// I/O Inputs              
	IN_MesAlarmPwr_IO		   : BOOL ;	              // (NA)[P,H,B] Remote control Power supply Error IO  	
	MesDataExd					: CB_Switch ; 		
END_VAR

VAR_OUTPUT
	
	//Child objects
	OUT_CmdOpen_IO	           : BOOL ; 	          // (NA) Physical I/O Open Command IO
	OUT_CmdClose_IO			   : BOOL ; 	          // (NA) Physical I/O Close Command IO
	
END_VAR


VAR
	
	//M_OPENCLOSE VARIABLES//

	//M_OPENCLOSE VARIABLES//	
	ParamTP_Open	 			: TP ;				(* (NA) Temporisation for Open pulse Command*)
	ParamTP_Close 				: TP ;				(* (NA) Temporisation for Close pulse Command	*)
		
END_VAR

METHOD M_AlarmManagement
//////////////////
// Manages Contactor alarms and warnings
/////////////////

VAR 
	// Method local variables (reinitialized at each cycle) 
	FB_AlarmCodeManager			: FB_AlarmCodeManager ; 

END_VAR
VAR_INPUT
	
END_VAR
// Check if command and measures are matching after tempo
FB_CheckCommand	(T:= ParamTimeOut_Close, bCmd:=OUT_CmdClose_IO , bMes := MesDataExd.MesData.MesClosed , bImpulsion := FALSE , bReset := CmdClearFault_G OR OUT_CmdClose_IO) ; 
FB_CheckCommand2(T:= ParamTimeOut_Open , bCmd:= OUT_CmdOpen_IO , bMes :=NOT MesDataExd.MesData.MesClosed , bImpulsion := FALSE , bReset := CmdClearFault_G OR OUT_CmdOpen_IO) ; 

TON_NotClosedAndNotOpened(IN:=  NOT MesClosed AND NOT MesOpened , PT := ParamTimeOut_Alarm) ; 
TON_ClosedAndOpened(IN:=MesClosed AND MesOpened, PT := ParamTimeOut_Alarm) ; 

// ALARM CODE //

	FB_AlarmCodeManager(
		bAlarm1			:= FALSE 	, 								// 
		bAlarm2			:= TON_NotClosedAndNotOpened.Q,					// Incoherent State measure (Not Opened and not Closed)
		bAlarm3 		:= TON_ClosedAndOpened.Q   , 					// Incoherent State measure (Opened and Closed)	
		bAlarm4			:= FB_CheckCommAND.bWarning , 					// Close command failed
		bAlarm5			:= FB_CheckCommand2.bWarning  , 				// Open Command failed
		bAlarm6			:= FALSE,                                   	//
		bAlarm7			:= FALSE,                                   	//
		bAlarm8			:= FALSE,                                   	//
		bAlarm9			:= FALSE,                                   	//
		bAlarm10		:= FALSE,                                   	//
		bAlarm11		:= FALSE,                                   	//
		bAlarm12		:= FALSE,                                   	//
		bAlarm13		:= FALSE,                                   	//
		bAlarm14		:= FALSE,                                   	//
		bAlarm15		:= FALSE , 										//
		wAlarmCode		=>MesDataExd.MesData.MesAlarmCode);

		

//WARNING CODE//
		FB_AlarmCodeManager(
		bAlarm1			:= FALSE,										//
		bAlarm2			:= FALSE,										//
		bAlarm3 		:= FALSE,										// 
		bAlarm4			:= MesDataExd.MesAlarmPwr, 						// Power supply fault
		bAlarm5			:= FALSE , //
		bAlarm6			:= FALSE , 
		bAlarm7			:=FALSE , //
		bAlarm8			:= FALSE, 										//
		bAlarm9			:= FALSE,                                       //
		bAlarm10		:= FALSE,                                       //
		bAlarm11		:= FALSE,                                       //
		bAlarm12		:= FALSE,                                       //
		bAlarm13		:= FALSE,                                       //
		bAlarm14		:= FALSE,                                       //
		bAlarm15		:= FALSE, 										//
		wAlarmCode 		=>MesDataExd.MesData.MesWarningCode);

// EVENT CODE //
	FB_AlarmCodeManager(
		bAlarm1			:= OUT_CmdOpen_IO, 								// Open Command
		bAlarm2			:= OUT_CmdClose_IO, 							// Close Command
		bAlarm3			:= MesOpened, 									// Opened Position
		bAlarm4			:= MesClosed, 									// Closed Position
		bAlarm5			:= IN_CmdReset, 								// Reset command
		bAlarm6			:= FALSE, 										//
		bAlarm7			:= FALSE,                   					//
		bAlarm8			:= FALSE,                   					//
		bAlarm9			:= FALSE,                   					//
		bAlarm10		:= FALSE,                   					//
		bAlarm11		:= FALSE,                   					//
		bAlarm12		:= FALSE,                   					//
		bAlarm13		:= FALSE, 										//
		bAlarm14		:= FALSE,                   					//
		bAlarm15		:= FALSE,                   					//
		wAlarmCode		=>MesDataExd.MesData.MesEventCode);   
                                           

MesDataExd.MesAlarmPwr		    := IN_MesAlarmPwr_IO ; 

MesDataExd.OUT_CmdClose		    := OUT_CmdClose_IO ; 
MesDataExd.OUT_CmdOpen		    := OUT_CmdOpen_IO ;
END_METHOD

METHOD M_Execute
VAR_INPUT
END_VAR

VAR

END_VAR

// PERMANENT CONDITIONS //	
MesDataExd.MesData.MesCP_Open					:= IN_CmdOpen AND NOT IN_CmdReset;
MesDataExd.MesData.MesCP_Close				:= NOT MesDataExd.MesData.MesClosed AND IN_CmdClose AND NOT MesDataExd.MesData.MesAlarmCode.0 AND NOT MesDataExd.MesData.MesCP_Open AND NOT IN_CmdReset ;


SUPER^.M_Execute();
END_METHOD

METHOD M_OpenClose
//////////////////
// Manages Opening and Closing of the contactor
//////////////////

VAR 
	// Method local variables (reinitialized at each cycle) 

	
END_VAR


// Open Command
ParamTP_Open(IN:= MesDataExd.MesData.MesCP_Open , PT:=ParamTP_Impulsion) ;
OUT_CmdOpen_IO	 := ParamTP_Open.Q ;                               			 // Impulsion that goes back to zero as soon as the state of the TP goes down. 

// Close Command
ParamTP_Close(IN:= MesDataExd.MesData.MesCP_Close , PT:=ParamTP_Impulsion) ;
OUT_CmdClose_IO	 := ParamTP_Close.Q ;                          			 // Impulsion that goes back to zero as soon as the state of the TP goes down.
END_METHOD

METHOD M_StateManager
//////////////////
// Manages Contactor State
/////////////////

VAR 
	// Method local variables (reinitialized at each cycle) 
	
END_VAR
MesState := 0 ; 
IF MesOpened THEN		// If the cell seems opens and closed in the same time, we will consider it as opened. 
	
	MesState.0 := 1 ; 
MesDataExd.MesData.MesClosed := FALSE ; 
MesDataExd.MesData.MesOpened := TRUE ; 
ELSIF MesClosed THEN
	
	MesState.1 := 1 ; 
MesDataExd.MesData.MesClosed := TRUE ; 
MesDataExd.MesData.MesOpened := FALSE ; 
ELSE 
	MesState.0 := 1 ;		// if the cell seems neither opened and neither closed , we will consider it as opened. 
MesDataExd.MesData.MesClosed := FALSE ; 	
MesDataExd.MesData.MesOpened := TRUE ; 
END_IF
END_METHOD

END_FUNCTION_BLOCK

// ---- 01_Equipement_Library/Batteries/FB_BAT_NARADA.TcPOU
FUNCTION_BLOCK FB_BAT_NARADA EXTENDS FB_BAT_Base

VAR_INPUT PERSISTENT
	
	//Com
	
		ParamIpAddress 			: STRING 	:='192.168.127.133' ; 		(* IP¨Address*)
		ParamUnitID				: BYTE  	:= 1 ; 					(* Modbus Unit ID*)
		ParamTcpPort			: UINT 		:= 502;					(* Modbus TCP Port*)

END_VAR

VAR_INPUT
	
	IN_CmdOpenDC						: BOOL;
	IN_CmdCloseDC 						: BOOL;

	MesDataExd							: BAT_NARADA;
	
END_VAR

VAR_OUTPUT

 	OUT_MesSoC_Min						: REAL;
    OUT_MesSoC_Max						: REAL;
	OUT_MesNbRackConnected				: REAL;
	OUT_MesEnomConnected				: REAL;
	OUT_MesSoCConnected					: REAL;

END_VAR


VAR
	
	//M_ALARM MANAGEMENT VARIABLES//
	
		CalModbusWriteAlarm			: BOOL;		// Modbus Write alarm
		ComWarning					: BOOL;		// Aggregated Communication warning
		ComAlarm					: BOOL;		// Aggregated communication Alarm
		
	//M_READ VARIABLES//
	
		// FB Read 
		
			ModbusReadInputRegs						: ARRAY[1..CstNbRack_BAT_G] OF FB_ModbusReadInputRegs;
			ModbusReadInputRegs1					: ARRAY[1..CstNbBms_BAT_G] OF FB_ModbusReadInputRegs;
			ModbusReadRegshvac						: ARRAY[1..4] OF FB_ModbusReadInputRegs;
			
		// Parameters FB Read
		
			// Alarms
			
			MesModbusReadAlarm_Racks 				: ARRAY[1..CstNbRack_BAT_G] OF BOOL ; 			// (NA) Modbus Read Alarm for all modbus frames		
			MesModbusReadAlarm_BMS 					: ARRAY[1..CstNbBms_BAT_G] OF BOOL ; 			// (NA) Modbus Read Alarm for all modbus frames	
			MesModbusReadAlarm 						: ARRAY[1..4] OF BOOL;
			// Regs
			
			MesModbusReadRegister					: ARRAY[1..CstNbRack_BAT_G] OF ARRAY[1..120] OF WORD;
			MesModbusReadInputRegister				: ARRAY[1..CstNbBms_BAT_G] OF ARRAY[1..120] OF WORD;
			MesModbusReadRegisterhvac				: ARRAY[1..CstNbBms_BAT_G] OF ARRAY[1..120] OF WORD;
			
			//Param
			
			ParamModbusHoldingRegisterFirst			: WORD	:= 16#1001;
			ParamModbusHoldingRRegisterRead			: WORD	:= 70;
			ParamModbusHoldingRegisterSecond		: WORD	:= 16#1100;
			ParamModbusHoldingRegisterReadSecond	: WORD	:= 32;
			
			ParamModbusRegisterFirst				: WORD	:= 16#2001;
			ParamModbusRegisterRead					: WORD	:= 31;
			ParamModbusRegisterNotRead				: WORD	:= 1201;
			ParamModbusRegisterRacksOffset			: WORD	:= 0;
			ParamModbusRegisterTotal				: WORD	:= 1231;
											
	//M_WRITE VARIABLES //  
	
		AX_Cmd	AT%Q* 								: ARRAY[1..3] OF WORD;
		AX_ModbusWrite								: ARRAY[1..4] OF FB_ModbusWriteSingleRegister;
		AX_bAlarmWrite								: ARRAY[1..4] OF BOOL;
		AX_uAlarmWrite								: ARRAY[1..4] OF UDINT ; 
		AX_ModbusWriteSingleRegister				: ARRAY[1..4] OF FB_ModbusWriteSingleRegister;
		AX_bAlarmWriteSingleRegister				: ARRAY[1..4] OF BOOL;
		AX_uAlarmWriteSingleRegister				: ARRAY[1..4] OF UDINT ; 
		Trig_CmdOpenDC								: R_TRIG;
		Trig_CmdCloseDC								: R_TRIG;
		Trig_CmdReset								: R_TRIG;
	
	//M_STATEMANAGER VARIABLES//
	//M_INIT VARIABLES //
	//M_EVALUATE VARIABLES //
	//M_EXECUTE VARIABLES//
		
	//Test//	
	
		Xtest				: BOOL;
		TrigStopBat			: BOOL := FALSE;
		xTestReal			: REAL;
		xTestInt			: INT;
		xTestWord			: WORD;
		CmdPCSStop			: BOOL;
		CmdPCSStart			: BOOL;
		
		
END_VAR

METHOD M_AlarmManagement
//////////////////
//  Battery Area  Alarm Management 
/////////////////

VAR 
	// Method local variables (reinitialized at each cycle) 
	FB_AlarmCodeManager 		: FB_AlarmCodeManager ; 
                            	
	KK							: UINT;				// For Loop 
	                 
END_VAR
//COMMUNICATION//
	
	//ComWarning 	:= ;
	ComAlarm	:= MesDataExd.MesBAUState.3;

	
	FOR KK:=1 TO ParamNbRacks DO // nb of trame = 4
	//	ComWarning 	:= ComWarning OR MesModbusReadAlarmRacks[KK][1] OR MesModbusReadAlarmRacks[KK][2] ;
		ComAlarm	:= ComAlarm OR MesDataExd.AX_Rack[KK].MesData.MesIDConnectAlarm.4 OR MesDataExd.AX_Rack[KK].MesData.MesIDConnectAlarm.5;
	END_FOR	
	
	//Warning
	MesDataExd.MesData.MesWarningCom := ComWarning ; 
	//Alarm
	TON_ComAlarm(IN:= ComAlarm , PT:= ParamTempoComAlarm, Q=>MesDataExd.MesData.MesAlarmCom) ;	// Alarms if ALL TRAM MODBUS did not work and timeout of 15s
	


TON_ComAlarm(IN:= ComAlarm , PT:= ParamTempoComAlarm, Q=>MesDataExd.MesData.MesAlarmCom) ;	// Alarms if ALL TRAM MODBUS did not work and timeout of 15s
	



	FB_AlarmCodeManager(	
		bAlarm1			:= MesDataExd.MesData.MesAlarmCom, 							// Com alarm
		bAlarm2			:= FALSE,													// 
		bAlarm3			:= FALSE, 													//                  
		bAlarm4			:= FALSE, 													//                      
		bAlarm5			:= FALSE, 													//                 
		bAlarm6			:= FALSE, 													//          
		bAlarm7			:= FALSE, 													//          
		bAlarm8			:= FALSE, 													//          
		bAlarm9			:= FALSE,   												//         
		bAlarm10		:= FALSE,   												//         
		bAlarm11		:= FALSE,   												//          
		bAlarm12		:= FALSE, 													//  						                
		bAlarm13		:= FALSE, 													//  						                 
		bAlarm14		:= FALSE, 													//  						                 
		bAlarm15		:= FALSE, 													//  						
		wAlarmCode		=> MesDataExd.MesData.MesAlarmCode);


// WARNING CODE //
	FB_AlarmCodeManager(	
		bAlarm1			:= MesDataExd.MesData.MesWarningCom, 						// Communication warning 
		bAlarm2			:= FALSE, 													//
		bAlarm3			:= FALSE, 													//
		bAlarm4			:= FALSE, 													//      
		bAlarm5			:= FALSE, 													//      
		bAlarm6			:= FALSE, 													//      
		bAlarm7			:= FALSE, 													//      
		bAlarm8			:= FALSE,   												//         
		bAlarm9			:= FALSE,   												//         
		bAlarm10		:= FALSE,   												//         
		bAlarm11		:= FALSE,   												//         
		bAlarm12		:= FALSE,   												//         
		bAlarm13		:= FALSE,  													//         
		bAlarm14		:= FALSE,  													//         
		bAlarm15		:= FALSE,	    											// 
		wAlarmCode		=> MesDataExd.MesData.MesWarningCode);          
		


// EVENT CODE //
	FB_AlarmCodeManager(
		bAlarm1			:= FALSE,													//
		bAlarm2			:= FALSE,													//
		bAlarm3			:= FALSE,													//
		bAlarm4			:= FALSE,													//		
		bAlarm5			:= IN_CmdOpenDC,                                            // Open DC command
		bAlarm6			:= IN_CmdCloseDC,                                           // Close DC Command
		bAlarm7			:= FALSE,                                                   //
		bAlarm8			:= FALSE,                                                   //
		bAlarm9			:= FALSE,                                                   //
		bAlarm10		:= FALSE,                                                   //
		bAlarm11		:= FALSE,                                                   //
		bAlarm12		:= FALSE,                                                   //
		bAlarm13		:= FALSE,                                                   //
		bAlarm14		:= FALSE,                                                   //
		bAlarm15		:= FALSE,                                                   //
		wAlarmCode		=> MesDataExd.MesData.MesEventCode);


	FB_AlarmCodeManager(	
        bAlarm1			:= MesDataExd.MesChargeStatus= 1,  									// Charge Status  -  OFF
        bAlarm2			:= MesDataExd.MesChargeStatus= 2,  									// Charge Status  -  EMPTY
        bAlarm3			:= MesDataExd.MesChargeStatus= 3,  									// Charge Status  -  DISCHARGING
        bAlarm4			:= MesDataExd.MesChargeStatus= 4,  									// Charge Status  -  CHARGING
        bAlarm5			:= MesDataExd.MesChargeStatus= 5,  									// Charge Status  -  FULL
        bAlarm6			:= MesDataExd.MesChargeStatus= 6,  									// Charge Status  -  HOLDING
        bAlarm7			:= MesDataExd.MesChargeStatus= 7,  									// Charge Status  -  TESTING
		bAlarm8			:= FALSE,                                                   //
		bAlarm9			:= FALSE,                                                   //
		bAlarm10		:= FALSE,                                                   //
		bAlarm11		:= FALSE,                                                   //
		bAlarm12		:= FALSE,                                                   //
		bAlarm13		:= FALSE,                                                   //
		bAlarm14		:= FALSE,                                                   //
		bAlarm15		:= FALSE,                                                   //
		wAlarmCode		=> MesDataExd.MesChargeStatus);

		

	FB_AlarmCodeManager(	
        bAlarm1			:= MesDataExd.MesData.MesIDState= 1,  				// State of the Battery Bank  -  DISCONNECTED
        bAlarm2			:= MesDataExd.MesData.MesIDState= 2,  				// State of the Battery Bank  -  INITIALIZING
        bAlarm3			:= MesDataExd.MesData.MesIDState= 3,  				// State of the Battery Bank  -  CONNECTED
        bAlarm4			:= MesDataExd.MesData.MesIDState= 4,  				// State of the Battery Bank  -  STANDBY
        bAlarm5			:= MesDataExd.MesData.MesIDState= 5,  				// State of the Battery Bank  -  SOC PROTECTION
        bAlarm6			:= MesDataExd.MesData.MesIDState= 6,  				// State of the Battery Bank  -  SUSPENDING
        bAlarm7			:= MesDataExd.MesData.MesIDState= 99,  			// State of the Battery Bank  -  FAULT
		bAlarm8			:= FALSE,                       //
		bAlarm9			:= FALSE,                       //
		bAlarm10		:= FALSE,                       //
		bAlarm11		:= FALSE,                       //
		bAlarm12		:= FALSE,                       //
		bAlarm13		:= FALSE,                       //
		bAlarm14		:= FALSE,                       //
		bAlarm15		:= FALSE,                       //
		wAlarmCode		=> MesDataExd.MesData.MesIDState
);


	FB_AlarmCodeManager(	
        bAlarm1		:= MesDataExd.MesData.MesEvt1.0,  			// Battery Event 1 -  COMMUNICATION_ERROR
        bAlarm2		:= MesDataExd.MesData.MesEvt1.1,  			// Battery Event 1 -  OVER_TEMP_ALARM
        bAlarm3		:= MesDataExd.MesData.MesEvt1.2,  			// Battery Event 1 -  OVER_TEMP_WARNING
        bAlarm4		:= MesDataExd.MesData.MesEvt1.3,  			// Battery Event 1 -  UNDER_TEMP_ALARM
        bAlarm5		:= MesDataExd.MesData.MesEvt1.4,  			// Battery Event 1 -  UNDER_TEMP_WARNING
        bAlarm6		:= MesDataExd.MesData.MesEvt1.5,  			// Battery Event 1 -  OVER_CHARGE_CURRENT_ALARM
        bAlarm7		:= MesDataExd.MesData.MesEvt1.6,  			// Battery Event 1 -  OVER_CHARGE_CURRENT_WARNING
        bAlarm8		:= MesDataExd.MesData.MesEvt1.7,  			// Battery Event 1 -  OVER_DISCHARGE_CURRENT_ALARM
        bAlarm9		:= MesDataExd.MesData.MesEvt1.8,  			// Battery Event 1 -  OVER_DISCHARGE_CURRENT_WARNING
        bAlarm10	:= MesDataExd.MesData.MesEvt1.9,  			// Battery Event 1 -  OVER_VOLT_ALARM
        bAlarm11	:= MesDataExd.MesData.MesEvt1.10,  		// Battery Event 1 -  OVER_VOLT_WARNING
        bAlarm12	:= MesDataExd.MesData.MesEvt1.11,  		// Battery Event 1 -  UNDER_VOLT_ALARM
        bAlarm13	:= MesDataExd.MesData.MesEvt1.12,  		// Battery Event 1 -  UNDER_VOLT_WARNING
        bAlarm14	:= MesDataExd.MesData.MesEvt1.13,  		// Battery Event 1 -  UNDER_SOC_MIN_ALARM
        bAlarm15	:= MesDataExd.MesData.MesEvt1.14,  		// Battery Event 1 -  UNDER_SOC_MIN_WARNING
		wAlarmCode	=> MesDataExd.MesData.MesAlarmCode_MesEvt1_1
);

	FB_AlarmCodeManager(	
        bAlarm1		:= MesDataExd.MesData.MesEvt1.15,  		// Battery Event 1 -  OVER_SOC_MAX_ALARM
        bAlarm2		:= MesDataExd.MesData.MesEvt1.16,  		// Battery Event 1 -  OVER_SOC_MAX_WARNING
        bAlarm3		:= MesDataExd.MesData.MesEvt1.17,  		// Battery Event 1 -  VOLTAGE_IMBALANCE_WARNING
        bAlarm4		:= MesDataExd.MesData.MesEvt1.18,  		// Battery Event 1 -  TEMPERATURE_IMBALANCE_ALARM
        bAlarm5		:= MesDataExd.MesData.MesEvt1.19,  		// Battery Event 1 -  TEMPERATURE_IMBALANCE_WARNING
        bAlarm6		:= MesDataExd.MesData.MesEvt1.20,  		// Battery Event 1 -  CONTACTOR_ERROR
        bAlarm7		:= MesDataExd.MesData.MesEvt1.21,  		// Battery Event 1 -  FAN_ERROR
        bAlarm8		:= MesDataExd.MesData.MesEvt1.22,  		// Battery Event 1 -  GROUND_FAULT
        bAlarm9		:= MesDataExd.MesData.MesEvt1.23,  		// Battery Event 1 -  OPEN_DOOR_ERROR
        bAlarm10	:= MesDataExd.MesData.MesEvt1.24,  		// Battery Event 1 -  CURRENT_IMBALANCE_WARNING
        bAlarm11	:= MesDataExd.MesData.MesEvt1.25,  		// Battery Event 1 -  OTHER_ALARM
        bAlarm12	:= MesDataExd.MesData.MesEvt1.26,  		// Battery Event 1 -  OTHER_WARNING
        bAlarm13	:= MesDataExd.MesData.MesEvt1.27,  		// Battery Event 1 -  RESERVED_1
        bAlarm14	:= MesDataExd.MesData.MesEvt1.28,  		// Battery Event 1 -  CONFIGURATION_ALARM
        bAlarm15	:= MesDataExd.MesData.MesEvt1.29,  		// Battery Event 1 -  CONFIGURATION_WARNING
		wAlarmCode	=> MesDataExd.MesData.MesAlarmCode_MesEvt1_2
);

	FB_AlarmCodeManager(	
        bAlarm1			:= MesDataExd.MesData.MesEvtVnd1.0,  		// Battery Vendor Event 1   -  Cell Over Voltage Warning   
        bAlarm2			:= MesDataExd.MesData.MesEvtVnd1.1,  		// Battery Vendor Event 1   -  Cell Under Voltage Warning  
        bAlarm3			:= MesDataExd.MesData.MesEvtVnd1.2,  		// Battery Vendor Event 1   -  Cell Voltage Imbalance      
        bAlarm4			:= MesDataExd.MesData.MesEvtVnd1.3,  		// Battery Vendor Event 1   -  Cell Over Voltage Alarm     
        bAlarm5			:= MesDataExd.MesData.MesEvtVnd1.4,  		// Battery Vendor Event 1   -  Cell Under Voltage Alarm    
        bAlarm6			:= MesDataExd.MesData.MesEvtVnd1.5,  		// Battery Vendor Event 1   -  Cell Voltage Imbalance Alarm
        bAlarm7			:= MesDataExd.MesData.MesEvtVnd1.6,  		// Battery Vendor Event 1   -  Cell Over Voltage Fault     
        bAlarm8			:= MesDataExd.MesData.MesEvtVnd1.7,  		// Battery Vendor Event 1   -  Cell Under Voltage Fault    
        bAlarm9			:= MesDataExd.MesData.MesEvtVnd1.8,  		// Battery Vendor Event 1   -  Cell Voltage Imbalance Fault
        bAlarm10		:= MesDataExd.MesData.MesEvtVnd1.9,  		// Battery Vendor Event 1   -  Over Temperature Fault      
        bAlarm11		:= MesDataExd.MesData.MesEvtVnd1.10,  	// Battery Vendor Event 1   -  Under Temperature Fault     
        bAlarm12		:= MesDataExd.MesData.MesEvtVnd1.11,  	// Battery Vendor Event 1   -  Temperature Imbalance Fault 
        bAlarm13		:= MesDataExd.MesData.MesEvtVnd1.12,  	// Battery Vendor Event 1   -  Over Voltage Fault          
        bAlarm14		:= MesDataExd.MesData.MesEvtVnd1.13,  	// Battery Vendor Event 1   -  Under Voltage Fault         
        bAlarm15		:= MesDataExd.MesData.MesEvtVnd1.14,  	// Battery Vendor Event 1   -  Over Charge Current Fault   
		wAlarmCode		=>MesDataExd.MesData.MesAlarmCode_MesEvtVnd1_1
);

	FB_AlarmCodeManager(	
        bAlarm1			:= MesDataExd.MesData.MesEvtVnd1.15,  	// Battery Vendor Event 1  -  Over Discharge Current Fault      
        bAlarm2			:= MesDataExd.MesData.MesEvtVnd1.16,  	// Battery Vendor Event 1  -  String Connection Failure         
        bAlarm3			:= MesDataExd.MesData.MesEvtVnd1.17,  	// Battery Vendor Event 1  -  RBMS to MBMS Communication Failure
        bAlarm4			:= MesDataExd.MesData.MesEvtVnd1.18,  	// Battery Vendor Event 1  -  Temperature Sensor Failure       
        bAlarm5			:= MesDataExd.MesData.MesEvtVnd1.19,  	// Battery Vendor Event 1  -  Main Relay Open Failure          
        bAlarm6			:= MesDataExd.MesData.MesEvtVnd1.20,  	// Battery Vendor Event 1  -  Bus Voltage Imbalance             
        bAlarm7			:= MesDataExd.MesData.MesEvtVnd1.21,  	// Battery Vendor Event 1  -  Fan Failure                       
        bAlarm8			:= MesDataExd.MesData.MesEvtVnd1.22,  	// Battery Vendor Event 1  -  Voltage Sensor Failure            
        bAlarm9			:= MesDataExd.MesData.MesEvtVnd1.23,  	// Battery Vendor Event 1  -  Insulation Detection Warning      
        bAlarm10		:= MesDataExd.MesData.MesEvtVnd1.24,  	// Battery Vendor Event 1  -  Insulation Detection Fault        
		bAlarm11		:= FALSE,                                                   //
		bAlarm12		:= FALSE,                                                   //
		bAlarm13		:= FALSE,                                                   //
		bAlarm14		:= FALSE,                                                   //
		bAlarm15		:= FALSE,                                                   //
		wAlarmCode		=> MesDataExd.MesData.MesAlarmCode_MesEvtVnd1_2
);
END_METHOD

METHOD M_CP
//////////////////
//  Permanent conditions 
/////////////////

VAR 
	// Method local variables (reinitialized at each cycle) 
	
END_VAR


SUPER^.M_CP() ; 




Trig_Cmd_Read(CLK:=IN_CmdToggleRead);
Trig_Cmd_Write(CLK:=IN_CmdToggleWrite);
	
IF Trig_Cmd_Read.Q THEN
	IN_CmdToggleRead := FALSE;
	MesDataExd.MesData.MesCP_Read := NOT MesDataExd.MesData.MesCP_Read;
END_IF


IF Trig_Cmd_Write.Q THEN
	IN_CmdToggleWrite := FALSE;
	MesDataExd.MesData.MesCP_Write := NOT MesDataExd.MesData.MesCP_Write;
END_IF
END_METHOD

METHOD M_Evaluate : BOOL
VAR_INPUT
END_VAR
VAR
	KK : UINT;
	
END_VAR

MesDataExd.MesData.MesSoC_Max :=0;
MesDataExd.MesData.MesSoC_Min :=0;
MesDataExd.MesSoCConnected:=0;
MesDataExd.MesNbRackConnected := 0;
MesDataExd.MesData.MesEnomConnected := 0;

FOR KK := 1 TO CstNbRack_BAT_G DO
		
	IF MesDataExd.AX_RACK[KK].MesData.MesIDState = 3 THEN
		
		IF MesDataExd.MesData.MesSoC_Min = 0 THEN
			
			MesDataExd.MesData.MesSoC_Min := MesDataExd.AX_RACK[KK].MesData.MesSoC;
			
		END_IF
		
		MesDataExd.MesData.MesSoC_Max := MAX(MesDataExd.MesData.MesSoC_Max, MesDataExd.AX_RACK[KK].MesData.MesSoC);
		MesDataExd.MesData.MesSoC_Min := MIN(MesDataExd.MesData.MesSoC_Min, MesDataExd.AX_RACK[KK].MesData.MesSoC);
		
	END_IF
	
	MesDataExd.MesNbRackConnected := MesDataExd.MesNbRackConnected + SEL(MesDataExd.AX_RACK[KK].MesData.MesIDState = 3, 0, 1);
	MesDataExd.MesData.MesEnomConnected := MesDataExd.MesData.MesEnomConnected + SEL(MesDataExd.AX_RACK[KK].MesData.MesIDState = 3, 0, ParamEnomRack) ;
	MesDataExd.MesSoCConnected := MesDataExd.MesSoCConnected + SEL(MesDataExd.AX_RACK[KK].MesData.MesIDState = 3, 0, MesDataExd.AX_RACK[KK].MesData.MesSoC);
	
END_FOR

MesDataExd.MesSoCConnected := SEL(MesDataExd.MesNbRackConnected>1 , 0 , MesDataExd.MesSoCConnected / MesDataExd.MesNbRackConnected ) ;

OUT_MesSoC_Min				:=		MesDataExd.MesData.MesSoC_Min;
OUT_MesSoC_Max				:=		MesDataExd.MesData.MesSoC_Max;
OUT_MesNbRackConnected		:=		MesDataExd.MesNbRackConnected;
OUT_MesEnomConnected		:=		MesDataExd.MesData.MesEnomConnected;	
OUT_MesSoCConnected			:=		MesDataExd.MesSoCConnected;
END_METHOD

METHOD M_Init
VAR 

END_VAR
END_METHOD

METHOD M_Read


VAR 

	KK			: DINT;

END_VAR


IF MesDataExd.MesData.MesCP_Read  THEN	

	// Acquisition données BMS
	
	ModbusReadInputRegs1[1]
		(
			pDestAddr 	:= ADR(MesModbusReadInputRegister[1]),
			sIPAddr 	:= ParamIpAddress,
			tTimeout 	:= ParamTimeout,
			nTcpPort 	:= 502,
			nQuantity 	:= ParamModbusHoldingRRegisterRead,
			nMBAddr 	:= ParamModbusHoldingRegisterFirst,
			cbLength 	:= SIZEOF(MesModbusReadInputRegister[1]),
			nUnitID		:= 1,
			ModbusReadAlarm => MesModbusReadAlarm_BMS[1] , 
			ClockRead	:= ClockRead
		);	
		
		MesDataExd.MesStatusConnectionProcess			:= WORD_TO_UINT(MesModbusReadInputRegister[1][1]);
		
		MesDataExd.MesSystemOperationState				:= WORD_TO_UINT(MesModbusReadInputRegister[1][6]);
		MesDataExd.MesSystemChargeState					:= WORD_TO_UINT(MesModbusReadInputRegister[1][7]);
		MesDataExd.MesBAUState 					:= WORD_TO_UINT(MesModbusReadInputRegister[1][8]);
		MesDataExd.MesIDRackWState 					:= WORD_TO_UINT(MesModbusReadInputRegister[1][9]);
		MesDataExd.MesIDRack						:= WORD_TO_UINT(MesModbusReadInputRegister[1][10]);
		MesDataExd.MesIDRackCriticalState				:= WORD_TO_UINT(MesModbusReadInputRegister[1][11]);
		                                                                                      
		MesDataExd.MesData.MesUdc						:= WORD_TO_UINT(MesModbusReadInputRegister[1][12])*0.1;
		MesDataExd.MesData.MesIdc						:=  WORD_TO_INT(MesModbusReadInputRegister[1][13])*0.1;
		MesDataExd.MesData.MesSoC						:= WORD_TO_UINT(MesModbusReadInputRegister[1][14])*0.1;
		MesDataExd.MesData.MesSoH						:= WORD_TO_UINT(MesModbusReadInputRegister[1][15])*0.1;
		MesDataExd.MesInsulation						:= WORD_TO_UINT(MesModbusReadInputRegister[1][16])*10;
		MesDataExd.MesData.MesECharge					:= WORD_TO_UINT(MesModbusReadInputRegister[1][17]);
		MesDataExd.MesData.MesEDischarge				:= WORD_TO_UINT(MesModbusReadInputRegister[1][18]);
		MesDataExd.MesData.MesCCL						:= WORD_TO_UINT(MesModbusReadInputRegister[1][19])*0.1;		
		MesDataExd.MesData.MesDCL						:= WORD_TO_UINT(MesModbusReadInputRegister[1][20])*0.1;
		MesDataExd.MesIdiff								:= WORD_TO_UINT(MesModbusReadInputRegister[1][21])*0.1;
		MesDataExd.MesUdiff								:=  WORD_TO_INT(MesModbusReadInputRegister[1][22])*0.1;	
		                                                                                      
		MesDataExd.MesIDRack_UdcMax_Cell  				:= WORD_TO_UINT(MesModbusReadInputRegister[1][23]);
		MesDataExd.MesIDModule_UdcMax_Cell 				:= WORD_TO_UINT(MesModbusReadInputRegister[1][24]);
		MesDataExd.MesIDCell_UdcMax		 				:= WORD_TO_UINT(MesModbusReadInputRegister[1][25]);
		MesDataExd.MesUdcMax_Cell						:= WORD_TO_UINT(MesModbusReadInputRegister[1][26])*0.001;	
	                                                                                          
		MesDataExd.MesIDRack_UdcMin_Cell  				:= WORD_TO_UINT(MesModbusReadInputRegister[1][27]);
		MesDataExd.MesIDModule_UdcMin_Cell 		 		:= WORD_TO_UINT(MesModbusReadInputRegister[1][28]);
		MesDataExd.MesIDCell_UdcMin		 				:= WORD_TO_UINT(MesModbusReadInputRegister[1][29]);
		MesDataExd.MesUdcMin_Cell    					:= WORD_TO_UINT(MesModbusReadInputRegister[1][30])*0.001;
                                                                                              
   		MesDataExd.MesUdc_Rack							:= WORD_TO_UINT(MesModbusReadInputRegister[1][31])*0.001;
                                                                                              
		MesDataExd.MesIDRack_TempMax_Cell       		:= WORD_TO_UINT(MesModbusReadInputRegister[1][32]); 
		MesDataExd.MesIDModule_TempMax_Cell           	:= WORD_TO_UINT(MesModbusReadInputRegister[1][33]); 
		MesDataExd.MesIDCell_TempMax           			:= WORD_TO_UINT(MesModbusReadInputRegister[1][34]);
		MesDataExd.MesTempMax_Cell               		:= 	WORD_TO_UINT(MesModbusReadInputRegister[1][35])*0.1;      	      	
		MesDataExd.MesIDRack_TempMin_Cell        		:= WORD_TO_UINT(MesModbusReadInputRegister[1][36]);      	
		MesDataExd.MesIDModule_TempMin_Cell     		:= WORD_TO_UINT(MesModbusReadInputRegister[1][37]); 
		MesDataExd.MesIDCell_TempMin           			:= WORD_TO_UINT(MesModbusReadInputRegister[1][38]); 
		MesDataExd.MesTempMin_Cell               		:=  WORD_TO_INT(MesModbusReadInputRegister[1][39])*0.1;     	
		MesDataExd.MesTemp_Racks                  		:= WORD_TO_UINT(MesModbusReadInputRegister[1][40])*0.1;     

	// Acquisition données racks 
	
	FOR KK := 1 TO ParamNbRacks DO
		ModbusReadInputRegs[KK]
		(
			pDestAddr 	:= ADR(MesModbusReadRegister[KK]),
			sIPAddr 	:= ParamIpAddress,
			tTimeout 	:= ParamTimeout,
			nTcpPort 	:= 502,
			nQuantity 	:= ParamModbusRegisterRead,
			nMBAddr 	:= ParamModbusRegisterFirst,
			cbLength 	:= SIZEOF(MesModbusReadRegister[KK]),
			nUnitID		:= DINT_TO_BYTE(KK+1),
			ModbusReadAlarm => MesModbusReadAlarm_Racks[KK] , 
			ClockRead	:= ClockRead
		);	
		
		
		MesDataExd.AX_Rack[KK].MesData.MesID_String							:= DINT_TO_WORD(KK);
		
		MesDataExd.AX_Rack[KK].MesNaradaIDState								:= WORD_TO_UINT(MesModbusReadRegister[KK][1]);
		                                                                                                 
		MesDataExd.AX_Rack[KK].MesData.MesIDState_DCSwitch					:= WORD_TO_UINT(MesModbusReadRegister[KK][3]);   
		MesDataExd.AX_Rack[KK].MesData.MesIDConnectAlarm					:= WORD_TO_UINT(MesModbusReadRegister[KK][4]);   
		MesDataExd.AX_Rack[KK].MesIDWarning									:= WORD_TO_UINT(MesModbusReadRegister[KK][5]);       
		MesDataExd.AX_Rack[KK].MesData.MesIDAlarm							:= WORD_TO_UINT(MesModbusReadRegister[KK][6]);         
		MesDataExd.AX_Rack[KK].MesIDCriticalAlarm							:= WORD_TO_UINT(MesModbusReadRegister[KK][7]);   
		MesDataExd.AX_Rack[KK].MesData.MesIDDisableReason					:= WORD_TO_UINT(MesModbusReadRegister[KK][8]);   
		
		MesDataExd.AX_Rack[KK].MesData.MesUdc                     			:= WORD_TO_UINT(MesModbusReadRegister[KK][11])*0.1;                                                                                                           
		MesDataExd.AX_Rack[KK].MesData.MesIdc                               := WORD_TO_UINT(MesModbusReadRegister[KK][12])*0.1;                            	               
		                                                                                                                 
		MesDataExd.AX_Rack[KK].MesData.MesSoC								:= WORD_TO_UINT(MesModbusReadRegister[KK][14])*0.1;   
		MesDataExd.AX_Rack[KK].MesData.MesSoH  								:= WORD_TO_UINT(MesModbusReadRegister[KK][15]);   
		
		MesDataExd.AX_Rack[KK].MesInsulationValue							:= WORD_TO_UINT(MesModbusReadRegister[KK][16])*10;   
		MesDataExd.AX_Rack[KK].MesPositiveInsulationValue					:= WORD_TO_UINT(MesModbusReadRegister[KK][17])*10;   
		MesDataExd.AX_Rack[KK].MesNegativeInsulationValue					:= WORD_TO_UINT(MesModbusReadRegister[KK][18])*10;   
        MesDataExd.AX_Rack[KK].MesCCL										:= WORD_TO_UINT(MesModbusReadRegister[KK][19])*0.1;   		
		MesDataExd.AX_Rack[KK].MesDCL										:= WORD_TO_UINT(MesModbusReadRegister[KK][20])*0.1;   
                                                                                         
		MesDataExd.AX_Rack[KK].MesData.MesIDModule_UdcMax_Cell				:= WORD_TO_UINT(MesModbusReadRegister[KK][21]);    
		MesDataExd.AX_Rack[KK].MesData.MesUdcMax_Cell 						:= WORD_TO_UINT(MesModbusReadRegister[KK][22])*0.001  ;
		MesDataExd.AX_Rack[KK].MesData.MesIDModule_UdcMin_Cell				:= WORD_TO_UINT(MesModbusReadRegister[KK][23]);    
		MesDataExd.AX_Rack[KK].MesData.MesUdcMin_Cell 						:= WORD_TO_UINT(MesModbusReadRegister[KK][24])*0.001  ; 
		MesDataExd.AX_Rack[KK].MesData.MesIDModule_TempMax_Module 			:= WORD_TO_UINT(MesModbusReadRegister[KK][25]);   
		MesDataExd.AX_Rack[KK].MesData.MesTempMax_Module          			:= WORD_TO_UINT(MesModbusReadRegister[KK][26])*0.1;   
		MesDataExd.AX_Rack[KK].MesData.MesIDModule_TempMin_Module 			:= WORD_TO_UINT(MesModbusReadRegister[KK][27]);   
		MesDataExd.AX_Rack[KK].MesData.MesTempMin_Module             		:= WORD_TO_UINT(MesModbusReadRegister[KK][28])*0.1;   
		MesDataExd.AX_Rack[KK].MesData.MesUdc_Cell		             		:= WORD_TO_UINT(MesModbusReadRegister[KK][29])*0.001;   
		MesDataExd.AX_Rack[KK].MesData.MesTemp_Module             			:= WORD_TO_UINT(MesModbusReadRegister[KK][30]);   

	END_FOR
	
	FOR KK:=1 TO 4 DO
		ModbusReadRegshvac[KK]
			(
				pDestAddr 	:= ADR(MesModbusReadRegisterhvac[KK]),
				sIPAddr 	:= ParamIpAddress,
				tTimeout 	:= ParamTimeout,
				nTcpPort 	:= 502,
				nQuantity 	:= ParamModbusHoldingRegisterReadSecond,
				nMBAddr 	:= DINT_TO_WORD(4352+37*(KK-1)),
				cbLength 	:= SIZEOF(MesModbusReadRegisterhvac[KK]),
				nUnitID		:= 1,
				ModbusReadAlarm =>MesModbusReadAlarm[KK] , 
				ClockRead	:= ClockRead
			);
			
		MesDataExd.AX_HVAC[KK].MesCoolTemp				:= WORD_TO_UINT(MesModbusReadRegisterhvac[KK][1]);	
		MesDataExd.AX_HVAC[KK].MesCoolSens				:= WORD_TO_UINT(MesModbusReadRegisterhvac[KK][2]);			
		MesDataExd.AX_HVAC[KK].MesHeatingTemp			:= WORD_TO_UINT(MesModbusReadRegisterhvac[KK][3]);	
		MesDataExd.AX_HVAC[KK].MesHeatingSens			:= WORD_TO_UINT(MesModbusReadRegisterhvac[KK][4]);	
		MesDataExd.AX_HVAC[KK].MesSetptHygro			:= WORD_TO_UINT(MesModbusReadRegisterhvac[KK][5]);	
		MesDataExd.AX_HVAC[KK].MesSensHygro				:= WORD_TO_UINT(MesModbusReadRegisterhvac[KK][6]);	
		MesDataExd.AX_HVAC[KK].MesTempmin				:= WORD_TO_UINT(MesModbusReadRegisterhvac[KK][7]);		
		MesDataExd.AX_HVAC[KK].MesTempmax				:= WORD_TO_UINT(MesModbusReadRegisterhvac[KK][8]);		
		MesDataExd.AX_HVAC[KK].MesHygromax				:= WORD_TO_UINT(MesModbusReadRegisterhvac[KK][9]);		
		MesDataExd.AX_HVAC[KK].MesState					:= WORD_TO_REAL(MesModbusReadRegisterhvac[KK][10]);		
		MesDataExd.AX_HVAC[KK].MesStateFanInternal		:= WORD_TO_BOOL(MesModbusReadRegisterhvac[KK][11]);	
		MesDataExd.AX_HVAC[KK].MesCompressorStatus 		:= WORD_TO_BOOL(MesModbusReadRegisterhvac[KK][12]);	
		MesDataExd.AX_HVAC[KK].MesHeating				:= WORD_TO_REAL(MesModbusReadRegisterhvac[KK][13]);			
		MesDataExd.AX_HVAC[KK].MesFrostTemp 			:= WORD_TO_BOOL(MesModbusReadRegisterhvac[KK][14]);			
		MesDataExd.AX_HVAC[KK].MesCondTemp				:= WORD_TO_BOOL(MesModbusReadRegisterhvac[KK][15]);			
		MesDataExd.AX_HVAC[KK].MesPressure1 			:= WORD_TO_UINT(MesModbusReadRegisterhvac[KK][16]);		
		MesDataExd.AX_HVAC[KK].MesTemp_Room				:= WORD_TO_UINT(MesModbusReadRegisterhvac[KK][17]);	
		MesDataExd.AX_HVAC[KK].MesHygro					:= WORD_TO_UINT(MesModbusReadRegisterhvac[KK][18]);
		MesDataExd.AX_HVAC[KK].MesTemp_Outside			:= WORD_TO_UINT(MesModbusReadRegisterhvac[KK][19]);                                    
		MesDataExd.AX_HVAC[KK].MesAlarmLow				:= WORD_TO_UINT(MesModbusReadRegisterhvac[KK][20]);	
		MesDataExd.AX_HVAC[KK].MesAlarmHigh				:= WORD_TO_UINT(MesModbusReadRegisterhvac[KK][21]);	
	END_FOR

END_IF
END_METHOD

METHOD M_StartStop
//////////////////
//  Start or stop BBMS via CAN bus   
/////////////////

VAR 
	// Method local variables (reinitialized at each cycle) 

END_VAR
END_METHOD

METHOD M_StateManager
//////////////////
// Detect which is the state of the PCS system . 
/////////////////

VAR 
	// Method local variables (reinitialized at each cycle) 
	KK : INT;

END_VAR



// MESA Creation Charge Status

    IF	MesDataExd.MesSystemOperationState = 4 THEN							
		MesDataExd.MesChargeStatus:= 1;  									// Charge Status  -  OFF
		
	ELSIF MesDataExd.MesSystemOperationState = 1 THEN
		MesDataExd.MesChargeStatus:= 2;  									// Charge Status  -  EMPTY				
		
	ELSIF MesDataExd.MesSystemChargeState = 1 THEN
        MesDataExd.MesChargeStatus:= 3;  									// Charge Status  -  DISCHARGING
		
	ELSIF MesDataExd.MesSystemChargeState = 2 THEN
        MesDataExd.MesChargeStatus:= 4;  									// Charge Status  -  CHARGING
		
	ELSIF MesDataExd.MesSystemOperationState = 1 THEN
		MesDataExd.MesChargeStatus:= 5;  									// Charge Status  -  FULL 
		 
	END_IF
	

// MESA Creation IDState

	IF MesDataExd.MesBAUState.0 = 1 THEN
		MesDataExd.MesData.MesIDState:= 99; 								// State of the Battery Bank  -  FAULT
		
	ELSIF MesDataExd.MesSystemChargeState = 0 THEN
		MesDataExd.MesData.MesIDState:= 4; 									// State of the Battery Bank  -  STANDBY
		
	ELSIF MesDataExd.MesStatusConnectionProcess = 2 THEN
		MesDataExd.MesData.MesIDState:= 3; 									// State of the Battery Bank  -  CONNECTED
		
		ELSIF MesDataExd.MesStatusConnectionProcess = 3 THEN
		MesDataExd.MesData.MesIDState:= 1; 									// State OF the Battery Bank  -  DISCONNECTED
		
	ELSIF MesDataExd.MesStatusConnectionProcess = 1 THEN
		MesDataExd.MesData.MesIDState:= 2; 									// State of the Battery Bank  -  INITIALIZING
		
	ELSIF MesDataExd.MesSystemOperationState = 2  THEN
		MesDataExd.MesData.MesIDState:= 5; 									// State OF the Battery Bank  -  SOC PROTECTION

	END_IF
	
// MESA Creation MesEvtVnd1

    //MesDataExd.MesData.MesEvtVnd1.0,  		// Battery Vendor Event 1   -  Cell Over Voltage Warning   
    //MesDataExd.MesData.MesEvtVnd1.1,  		// Battery Vendor Event 1   -  Cell Under Voltage Warning  
    //MesDataExd.MesData.MesEvtVnd1.2,  		// Battery Vendor Event 1   -  Cell Voltage Imbalance      
    MesDataExd.MesData.MesEvtVnd1.3 := MesDataExd.MesIDRackWState.2; 		// Battery Vendor Event 1   -  Cell Over Voltage Alarm     
    MesDataExd.MesData.MesEvtVnd1.4 := MesDataExd.MesIDRackWState.3;   	// Battery Vendor Event 1   -  Cell Under Voltage Alarm    
    //MesDataExd.MesData.MesEvtVnd1.5,  		// Battery Vendor Event 1   -  Cell Voltage Imbalance Alarm
    MesDataExd.MesData.MesEvtVnd1.6 := MesDataExd.MesIDRack.2; 	// Battery Vendor Event 1   -  Cell Over Voltage Fault     
    MesDataExd.MesData.MesEvtVnd1.7 := MesDataExd.MesIDRack.3;  	// Battery Vendor Event 1   -  Cell Under Voltage Fault    
    //MesDataExd.MesData.MesEvtVnd1.8,  		// Battery Vendor Event 1   -  Cell Voltage Imbalance Fault
    //MesDataExd.MesData.MesEvtVnd1.9,  		// Battery Vendor Event 1   -  Over Temperature Fault      
    //MesDataExd.MesData.MesEvtVnd1.10,  	// Battery Vendor Event 1   -  Under Temperature Fault     
    //MesDataExd.MesData.MesEvtVnd1.11,  	// Battery Vendor Event 1   -  Temperature Imbalance Fault 
    //MesDataExd.MesData.MesEvtVnd1.12,  	// Battery Vendor Event 1   -  Over Voltage Fault          
    //MesDataExd.MesData.MesEvtVnd1.13,  	// Battery Vendor Event 1   -  Under Voltage Fault         
    //MesDataExd.MesData.MesEvtVnd1.14,  	// Battery Vendor Event 1   -  Over Charge Current Fault      
    //MesDataExd.MesData.MesEvtVnd1.15,  	// Battery Vendor Event 1  -  Over Discharge Current Fault      
    //MesDataExd.MesData.MesEvtVnd1.16,  	// Battery Vendor Event 1  -  String Connection Failure         
    //MesDataExd.MesData.MesEvtVnd1.17,  	// Battery Vendor Event 1  -  RBMS to MBMS Communication Failure
    //MesDataExd.MesData.MesEvtVnd1.18,  	// Battery Vendor Event 1  -  Temperature Sensor Failure       
    //MesDataExd.MesData.MesEvtVnd1.19,  	// Battery Vendor Event 1  -  Main Relay Open Failure          
    //MesDataExd.MesData.MesEvtVnd1.20,  	// Battery Vendor Event 1  -  Bus Voltage Imbalance             
    //MesDataExd.MesData.MesEvtVnd1.21,  	// Battery Vendor Event 1  -  Fan Failure                       
    //MesDataExd.MesData.MesEvtVnd1.22,  	// Battery Vendor Event 1  -  Voltage Sensor Failure            
    //MesDataExd.MesData.MesEvtVnd1.23,  	// Battery Vendor Event 1  -  Insulation Detection Warning      
    //MesDataExd.MesData.MesEvtVnd1.24,  	// Battery Vendor Event 1  -  Insulation Detection Fault        
	
// MESA Creation MesEvt1 

	MesDataExd.MesData.MesEvt1.0 := MesDataExd.MesBAUState.3; 			// Battery Event 1 -  COMMUNICATION_ERROR
	MesDataExd.MesData.MesEvt1.1 := MesDataExd.MesIDRack.6 OR MesDataExd.MesIDRack.8;			// Battery Event 1 -  OVER_TEMP_ALARM
	MesDataExd.MesData.MesEvt1.2 := MesDataExd.MesIDRackWState.6;			// Battery Event 1 -  OVER_TEMP_WARNING
	MesDataExd.MesData.MesEvt1.3 := MesDataExd.MesIDRack.7 OR MesDataExd.MesIDRack.9;			// Battery Event 1 -  UNDER_TEMP_ALARM
	MesDataExd.MesData.MesEvt1.4 := MesDataExd.MesIDRackWState.7; 			// Battery Event 1 -  UNDER_TEMP_WARNING
	MesDataExd.MesData.MesEvt1.5 := MesDataExd.MesIDRack.5;			// Battery Event 1 -  OVER_CHARGE_CURRENT_ALARM
	MesDataExd.MesData.MesEvt1.6 := MesDataExd.MesIDRackWState.5;			// Battery Event 1 -  OVER_CHARGE_CURRENT_WARNING
	MesDataExd.MesData.MesEvt1.7 := MesDataExd.MesIDRack.4;			// Battery Event 1 -  OVER_DISCHARGE_CURRENT_ALARM
	MesDataExd.MesData.MesEvt1.8 := MesDataExd.MesIDRackWState.4;			// Battery Event 1 -  OVER_DISCHARGE_CURRENT_WARNING
	MesDataExd.MesData.MesEvt1.9 := MesDataExd.MesIDRack.0;			// Battery Event 1 -  OVER_VOLT_ALARM
	MesDataExd.MesData.MesEvt1.10 := MesDataExd.MesIDRackWState.0;  		// Battery Event 1 -  OVER_VOLT_WARNING
	MesDataExd.MesData.MesEvt1.11 := MesDataExd.MesIDRack.1; 			// Battery Event 1 -  UNDER_VOLT_ALARM
	MesDataExd.MesData.MesEvt1.12 := MesDataExd.MesIDRackWState.1; 		// Battery Event 1 -  UNDER_VOLT_WARNING
	//MesData.MesEvt1.13  		// Battery Event 1 -  UNDER_SOC_MIN_ALARM
	//MesData.MesEvt1.14  		// Battery Event 1 -  UNDER_SOC_MIN_WARNING
	//MesData.MesEvt1.15  		// Battery Event 1 -  OVER_SOC_MAX_ALARM
	//MesData.MesEvt1.16  		// Battery Event 1 -  OVER_SOC_MAX_WARNING
	MesDataExd.MesData.MesEvt1.17 := MesDataExd.MesBAUState.4;			// Battery Event 1 -  VOLTAGE_IMBALANCE_WARNING
	//MesData.MesEvt1.18  		// Battery Event 1 -  TEMPERATURE_IMBALANCE_ALARM
	//MesData.MesEvt1.19  		// Battery Event 1 -  TEMPERATURE_IMBALANCE_WARNING
	//MesData.MesEvt1.20  		// Battery Event 1 -  CONTACTOR_ERROR
	//MesData.MesEvt1.21  		// Battery Event 1 -  FAN_ERROR
	MesDataExd.MesData.MesEvt1.22  :=  MesDataExd.MesIDRack.10; 		// Battery Event 1 -  GROUND_FAULT
	//MesData.MesEvt1.23  		// Battery Event 1 -  OPEN_DOOR_ERROR
    MesDataExd.MesData.MesEvt1.24 := MesDataExd.MesBAUState.5;			// Battery Event 1 -  CURRENT_IMBALANCE_WARNING
    //MesData.MesEvt1.25  		// Battery Event 1 -  OTHER_ALARM
    //MesData.MesEvt1.26  		// Battery Event 1 -  OTHER_WARNING
    //MesData.MesEvt1.27  		// Battery Event 1 -  RESERVED_1
    //MesData.MesEvt1.28  		// Battery Event 1 -  CONFIGURATION_ALARM
    //MesData.MesEvt1.29  		// Battery Event 1 -  CONFIGURATION_WARNING



MesDataExd.MesData.MesState.0 := MesDataExd.MesNbRackConnected = 0 ;
MesDataExd.MesData.MesState.1 :=   MesDataExd.MesNbRackConnected > 0 ;
END_METHOD

METHOD M_Write
VAR_INPUT
END_VAR
VAR
	InputAddr: WORD;
	RTCWord: ARRAY[1..6] OF BYTE;
	TriggerRTC: BOOL;

	KK : INT;
	MBWr: INT;
	

END_VAR
Trig_CmdCloseDC(CLK := IN_CmdCloseDC);//IN_CmdCloseDC);
Trig_CmdOpenDC(CLK := IN_CmdOpenDC);//IN_CmdOpenDC);

	IF Trig_CmdCloseDC.Q THEN
		IN_CmdCloseDC := FALSE;
		AX_Cmd[1] := 16#0001;
	END_IF
	IF Trig_CmdOpenDC.Q THEN
		IN_CmdOpenDC := FALSE;
		AX_Cmd[1] := 16#0002;
	END_IF

	AX_ModbusWriteSingleRegister[1]	// Close / Open DC 
		(
			InputWord	:= AX_Cmd[1],
			sIPAddr 	:= ParamIpAddress,
			tTimeout 	:= ParamTimeout,
			nTCPport 	:= ParamTcpPort,
			nMBAddr 	:= 16#0001,
			nUnitID 	:= ParamUnitID,
			WriteCmd 	:= MesDataExd.Mesdata.MesCP_Write AND (Trig_CmdOpenDC.Q OR Trig_CmdCloseDC.Q),
			ModbusWriteAlarm => AX_bAlarmWriteSingleRegister[1],
			ErrorId		=> AX_uAlarmWriteSingleRegister[1]
		);

	Trig_CmdReset(CLK := IN_CmdReset);

	IF Trig_CmdReset.Q THEN			// lacth the fault date of events. WE HAVE TO CHECK FIRST THE FAULT BEFORE DOING IT/ 
		IN_CmdReset := FALSE;
	END_IF

	AX_ModbusWriteSingleRegister[2]	// Reset 
		(
			InputWord	:= 1,
			sIPAddr 	:= ParamIpAddress,
			tTimeout 	:= ParamTimeout,
			nTCPport 	:= ParamTcpPort,
			nMBAddr 	:= 16#0009,
			nUnitID 	:= ParamUnitID,
			WriteCmd 	:= Trig_CmdReset.Q AND MesDataExd.Mesdata.MesCP_Write,
			ModbusWriteAlarm => AX_bAlarmWriteSingleRegister[2],
			ErrorId		=> AX_uAlarmWriteSingleRegister[2]
		);
	
	FOR KK := 2 TO ParamNbRacks + 1 DO
		
		AX_ModbusWriteSingleRegister[2]	// Reset 
			(
				InputWord	:= 1,
				sIPAddr 	:= ParamIpAddress,
				tTimeout 	:= ParamTimeout,
				nTCPport 	:= ParamTcpPort,
				nMBAddr 	:= 16#3201,
				nUnitID 	:= ParamUnitID,
				WriteCmd 	:= Trig_CmdReset.Q AND MesDataExd.Mesdata.MesCP_Write,
				ModbusWriteAlarm => AX_bAlarmWriteSingleRegister[2],
				ErrorId		=> AX_uAlarmWriteSingleRegister[2]
			);
	
	END_FOR
	
//Trig_Watchdog(CLK := CalLocalTimeStruct.wMilliseconds < 500 );	// watchdog every 5 seconds . 
//
//AX_ModbusWrite[3]	// Heartbeat 
//(
//	InputWord	:= CalLocalTimeStruct.wSecond,
//	sIPAddr 	:= ParamIpAddress,
//	tTimeout 	:= ParamTimeout,
//	nTCPport 	:= ParamTcpPort,
//	nMBAddr 	:= 20,
//	nUnitID 	:= ParamUnitID,
//	WriteCmd 	:= Trig_Watchdog.Q AND MesDataExd.Mesdata.MesCP_Write,
//	ModbusWriteAlarm => AX_bAlarmWrite[3],
//	ErrorId		=> AX_uAlarmWrite[3]
//);
END_METHOD

END_FUNCTION_BLOCK

// ---- 01_Equipement_Library/Batteries/FB_BAT_Base.TcPOU
FUNCTION_BLOCK FB_BAT_Base

VAR_INPUT PERSISTENT
	// Parameters of the Object (instance specific) 
	ParamTempoComAlarm				: TIME 		:= T#15S ; 				(* (s) Config : Tempo to detect LOC Alarm*)
	ParamTimeOutStart           	: TIME 		:= T#1M ;				(* (s) Config : Tempo to start before Timeout warning*)
	ParamTimeOutStop        		: TIME 		:= T#30S ;				(* (s) Config : Tempo to start before Timeout warning*)
                                	
	ParamEnomRack					: REAL 		:= 76.1904 ;  	  	(* (kWh) Nominal Energy Capacity of one Rack *)
	                            	
	ParamClockReadTime 				: TIME 		:= TIME#1S;	  			(* (Time) Read Modbus Frequency .   *)
	ParamClockWriteTime 			: TIME 		:= TIME#1S;   			(* (Time) Write Modbus Frequency .         *)
	ParamTimeout					: TIME  	:= T#1S ;		  			(* (Time) Timeout for modbus reading*)
	ParamTimeWatchdog				: TIME 		:= T#3S;						(* (Time) Time after which a fixed watchdog raises an alarm*)
	                            	
	                            	
	ParamNbRacks					: BYTE 	:= 12 ; 					(* (NA) Number of racks controlled .*)
	ParamEssNum						: UINT 	:= 1;						(* (NA) ID number of the SystemBms' father PCS*)
	ParamSystemBmsNum				: BYTE 	:= 1;						(* Ctrl Bat Index in case of several CtrlBat 						*)
                                	
END_VAR
VAR_INPUT
	IN_CmdReset					: BOOL;
    IN_CmdToggleRead				: BOOL;
    IN_CmdToggleWrite				: BOOL;
	
	IN_CmdStart					: BOOL;									// (NA) [P,H] External Start Command
	IN_CmdStop 					: BOOL; 								// (NA) [P,H] External Stop CommAND  
	
	
	
END_VAR

VAR_OUTPUT
	//Child objects
		
END_VAR

VAR
	//M_ALARMMANAGEMENT VARIABLES//
		TON_ComAlarm				: TON ; 								// Tempo before deteting loss of communication. 
		TON_ComWarning				: TON ; 								// Tempo before deteting loss of communication. 
		TON_WatchdogWarning			: TON ; 								// Tempo before deteting loss of communication. 
                                                        					
                                                        					
		                                                					
		MesComWarning				: BOOL ; 								// (NA) [P,H]  True if bad communication or LOC with at least one rack
		MesComAlarm					: BOOL ;								// True if complete loss of communication with BBMS 			
		CmdAlarmIntervention		: BOOL ; 								// (NA) Command Alarm in case of intervention
		Watchdog_Old				: BOOL ;
		
	//M_READ VARIABLES//
	///MesDataExd.MesData.acks				: ARRAY [1..CstNbRack_BBMS] OF RACK ; 	// (NA) [H,B] 	Racks  Data Structure  

//	MesDataExd		AT%Q*	: BAT ;							// (NA) [P,H,B] CTRLbat  Data Structure
		Trig_Cmd_Read				: R_TRIG;                                                                                        
		Trig_Cmd_Write				: R_TRIG;                                                                                        
	
	//M_CONNECT VARIABLES// 
		FB_CheckCommand1			: FB_CheckCommand ; 					// (NA) Functionnal Block to check if Connect Writing Successful
		FB_CheckCommand2			: FB_CheckCommand ;						// (NA) Functionnal Block to check if Disconnect  Writing Successful
	                                                            			

		CalCompareWarningConnect	: BOOL ;								// (NA) Connect failed alarm
		CalCompareWarningDisconnect	: BOOL ;								// (NA) Disconnect failed alarm
		                                                        			
	//M_STATEMANAGER VARIABLES//                                			
		FB_OperationIndex			: FB_OperationIndex ;       			
		CalLastStart				: STRING ;			 					// Datetime of the last Start
		                                                        			
		CalRunningTime				: INT ; 								// Total Running Time
		CalNbMove					: WORD ;								// Total Number of Start;
		                                                        			
		MesState 					: BYTE ; 								// (NA) [P,H,B]  Bit 0: Disconnected , Bit 1 : Ready, Bit 2 : Connected
		                                                        			
	//M_INIT VARIABLES //                                       			
		bInit						: BOOL := TRUE ; 						// (NA) Initialize object parameters at first cycle 
	                                                            			
	//M_EXECUTE VARIABLES//                                     			
		TP1							: TP ; 									// (NA) Tempo to define Modbus Reading Frequency 
		TP2 						: TP ; 									// (NA) Tempo to define Modbus Writing Frequency
		ClockRead					: BOOL;									// (NA) Modbus reading Clock
		ClockWrite 					: BOOL;									// (NA) Modbus writing Clock 	

END_VAR

METHOD M_AlarmManagement
//////////////////
//  Battery Area  Alarm Management 
/////////////////

VAR 
	// Method local variables (reinitialized at each cycle) 

END_VAR
END_METHOD

METHOD M_CP
//////////////////
//  Permanent conditions 
/////////////////

VAR 
	// Method local variables (reinitialized at each cycle) 
	
END_VAR
END_METHOD

METHOD M_Evaluate : BOOL
VAR_INPUT
END_VAR
END_METHOD

METHOD M_Execute
//////////////////
//  Method Calls 
/////////////////

VAR 
	// Method local variables (reinitialized at each cycle) 
	KK		: INT;

	MesModbusReadAlarm: INT;
END_VAR
// READING AND WRITING CLOCK //
	TP1(IN:=NOT TP1.Q , PT:= ParamClockReadTime);
	ClockRead 	:= TP1.Q ;
	
	TP2(IN:=NOT TP2.Q , PT:= ParamClockWriteTime);
	ClockWrite 	:= TP2.Q;	
	
// PERMANENT CONDITIONS //
	M_CP() ; 

// METHODS CALLS//
	IF bInit THEN
		M_Init() ; 
		bInit	:= FALSE ; 
	ELSIF CmdInit_G  OR IN_CmdReset THEN 
		bInit:= TRUE ;
	END_IF
	
	M_Read();
	
	M_Evaluate();
		
	M_StateManager() ; 
	M_Write();
	M_StartStop() ; 
	

	
	M_AlarmManagement();
END_METHOD

METHOD M_Init
VAR 

END_VAR
END_METHOD

METHOD M_Read
//////////////////
//  Read Modbus Variable for racks and BBMS .  
/////////////////

VAR 
	// Method local variables (reinitialized at each cycle) 

	
END_VAR
END_METHOD

METHOD M_StartStop
//////////////////
//  Read Modbus Variable for racks and BBMS .  
/////////////////

VAR 
	// Method local variables (reinitialized at each cycle) 

	
	ParamTimeOutCurtail: TIME;
END_VAR
END_METHOD

METHOD M_StateManager
//////////////////
// Detect which is the state of the PCS system . 
/////////////////

VAR 
	// Method local variables (reinitialized at each cycle) 

	
END_VAR
END_METHOD

METHOD M_Write
VAR_INPUT
END_VAR
VAR
	AX_ADDR 	: ARRAY[1..1] OF UINT := [1];
	AX_QTY		: ARRAY[1..1] OF BYTE := [3];
	AX_UnitID	: ARRAY[1..1] OF BYTE := [1];
END_VAR
END_METHOD

END_FUNCTION_BLOCK

// ---- 01_Equipement_Library/Batteries/FB_BAT_Sams.TcPOU
FUNCTION_BLOCK FB_BAT_Sams EXTENDS FB_BAT_Base
// SAMSUNG System BMS P3
VAR_INPUT PERSISTENT
		ParamIpAddress 					: STRING 	:='192.168.1.51' ; 
		ParamUnitID						: BYTE  	:= 1 ; 
		ParamTcpPort					: UINT 		:= 502;
		ParamReadAlarmTime				: TIME 		:= T#1M30S;
		ParamReadWarningTime			: TIME		:= T#30S;
		ParamNbRackString				: BYTE		:=1  ; // Nb of strings of module per racks . 
		ParamNbReadAtOnce				: BYTE		:=10 ; // Number of racks read at the same time . 
		ParamClockReadRack_Delay		: TIME 		:= T#500MS ; 			// Delay after bbms read and before rack read
		ParamEnom_Rack					: REAL 		:= 97;
END_VAR

VAR_INPUT
	
		IN_CmdOpenDC					: BOOL;
		IN_CmdCloseDC 					: BOOL;
		
		
		
		MesDataExd							: BAT_SAMS;
END_VAR

VAR_OUTPUT
	//Child objects
		
END_VAR

VAR
	//M_ALARMMANAGEMENT VARIABLES//
	
		MesRackAlarmCode				: WORD ;
		MesRackAlarmCode2				: WORD ;
		MesRackWarningCode				: WORD ;
		MesRackWarningCode2				: WORD ; 
		TON_BatteriesCharging			: TON ;
		TON_BatteriesDischarging		: TON ;
		
		AX_AlarmWords						: ARRAY[1..75] OF ST_ValuesAlarms;
		AX_AlarmWords_Null					: ARRAY[1..75] OF ST_ValuesAlarms;
		NumAlarmsActive						: UINT;
		
	//M_READ VARIABLES//
		ModbusRead						: FB_ModbusReadInputRegs ; 
		ModbusReadrack					: ARRAY[1..40] OF FB_ModbusReadInputRegs ; 
                     			
		MesBlock1_Temp					: ARRAY[0..119] OF WORD ; 	
		MesBlock2_Temp					: ARRAY[1..40] OF ARRAY[0..119] OF WORD ; 
		
		MesModbusReadAlarm				: BOOL;	
		MesModbusReadAlarmID			: UDINT;
		MesModbusReadAlarm2				: ARRAY[1..40] OF BOOL;	
		MesModbusReadAlarmID2			: ARRAY[1..40] OF UDINT;		

		CTU_ClockRead								: CTU ; 
		TON_ClockRead					: TON;
	
	//M_WRITE VARIABLES //
		AX_Cmd					AT%Q*	: ARRAY[1..3] OF WORD;
		AX_ModbusWrite					: ARRAY[1..3] OF FB_ModbusWriteSingleRegister;
		A1_ModbusWriteRTC				: FB_ModbusWrite ; 
		
		Trig_Watchdog					: R_TRIG;
		Trig_CmdOpenDC					: R_TRIG;
		Trig_CmdCloseDC					: R_TRIG;
		Trig_CmdReset					: R_TRIG;
		
	

	//M_STATEMANAGER VARIABLES//
	
	//M_INIT VARIABLES //
	
	//M_EVALUATE VARIABLES //
		Trig_NewDay						: R_TRIG;
		Trig_Second						: R_TRIG;
		
	//M_EXECUTE VARIABLES//
		AX_DFV 							: ARRAY[1..13] OF FB_DetectFixedValue;	

END_VAR

METHOD M_AlarmManagement
//////////////////
//  Battery Area  Alarm Management 
/////////////////

VAR 
	// Method local variables (reinitialized at each cycle) 
	FB_AlarmCodeManager 		: FB_AlarmCodeManager ; 
                            	
	KK							: UINT;				// For Loop 
	LL							: UINT;
	                        	
	ComWarning					: BOOL;				// Aggregated communication warning
	ComAlarm					: BOOL;				// Aggregated communication Alarm
	CalLOCRBMS					: BOOL;				// Lost of Communication (LOC) between BBMS and RBMS . 
	
	CalRackWarningSynthesis		: BOOL;
	CalRackAlarmSynthesis		: BOOL;

	MesSyntheseAlarmStatus		: WORD;
	MesNbMots					: UINT;
	WordTest					: WORD;
	ID_Journal					: UINT;
END_VAR

TON_ComWarning( in := MesModbusReadAlarm OR MesModbusReadAlarm2[1] OR MesModbusReadAlarm2[2] OR MesModbusReadAlarm2[3] OR MesModbusReadAlarm2[4] OR MesModbusReadAlarm2[5] OR MesModbusReadAlarm2[6] OR MesModbusReadAlarm2[7], PT := ParamReadWarningTime);
TON_ComAlarm(IN:=  MesModbusReadAlarm AND MesModbusReadAlarm2[1] AND MesModbusReadAlarm2[2]AND MesModbusReadAlarm2[3]AND MesModbusReadAlarm2[4]AND MesModbusReadAlarm2[5]AND MesModbusReadAlarm2[6]AND MesModbusReadAlarm2[7], PT := ParamReadAlarmTime);
MesComWarning := TON_ComWarning.Q;


MesDataExd.MesData.MesAlarmCom := TON_ComAlarm.Q;
	
// ALARM CODE //
	FB_AlarmCodeManager(	
		bAlarm1			:= MesDataExd.MesData.MesAlarmCom, 									// Com alarm
		bAlarm2			:= AX_DFV[13].OUT_bStatic,									// Watchdog alarm
		bAlarm3			:= MesDataExd.MesRackProtection1 >0 ,  						// Rack Protection Synthesis  1                    
		bAlarm4			:= MesDataExd.MesRackProtection2 >0  ,  						// Rack Protection Synthesis  2                        
		bAlarm5			:= MesDataExd.MesRackStringProtection1 >0 , 					// RackStringProtection Synthesis 1               
		bAlarm6			:= MesDataExd.MesRackStringProtection2 >0 , 					// RackStringProtection Synthesis 2
		bAlarm7			:= MesDataExd.MesRackStringProtection3 >0  , 					// RackStringProtection Synthesis 3   
		bAlarm8			:= MesDataExd.MesRackStringProtection4 >0  , 					// RackStringProtection Synthesis 4   
		bAlarm9			:= MesDataExd.MesAlarm1 >0 , 				  					// System Alarm 1               
		bAlarm10		:= MesDataExd.MesAlarm2 >0 , 	 								// System Alarm 2               
		bAlarm11		:= FALSE , 													//  						                
		bAlarm12		:= FALSE , 													//  						                
		bAlarm13		:= FALSE , 													//  						                 
		bAlarm14		:= FALSE , 													//  						                 
		bAlarm15		:= FALSE , 													//  						
		wAlarmCode		=>MesDataExd.MesData.MesAlarmCode);


// WARNING CODE //
	FB_AlarmCodeManager(	
		bAlarm1			:= MesComWarning, 											// Communication warning 
		bAlarm2			:= MesDataExd.MesRackAlarm1 >0,								// Rack Warning Synthesis 1                 
		bAlarm3			:= MesDataExd.MesRackAlarm2 >0,								// Rack Warning Synthesis 2                  
		bAlarm4			:= MesDataExd.MesRackStringAlarm1 >0 ,  						// Rack String Warning Synthesis 1                    
		bAlarm5			:= MesDataExd.MesRackStringAlarm2 >0,  						// Rack String Warning Synthesis 2                    
		bAlarm6			:= MesDataExd.MesRackStringAlarm3 >0,  						// Rack String Warning Synthesis 3                    
		bAlarm7			:= MesDataExd.MesRackStringAlarm4 >0,   						// Rack String Warning Synthesis 4                    
		bAlarm8			:= FALSE,   												//         
		bAlarm9			:= FALSE,   												//         
		bAlarm10		:= FALSE,   												//         
		bAlarm11		:= FALSE,   												//         
		bAlarm12		:= FALSE,   												//         
		bAlarm13		:= FALSE,  													//         
		bAlarm14		:= FALSE,  													//         
		bAlarm15		:= FALSE,	    											// 
		wAlarmCode		=>MesDataExd.MesData.MesWarningCode);          
		


TON_BatteriesCharging(IN := MesDataExd.MesSystemMode.15, PT := T#30S);
TON_BatteriesDischarging(IN := MesDataExd.MesSystemMode.14, PT := T#30S);


// EVENT CODE //
	FB_AlarmCodeManager(
		bAlarm1			:= TON_BatteriesCharging.Q ,								//Batteries charging
		bAlarm2			:= TON_BatteriesDischarging.Q,								//Batteries discharging
		bAlarm3			:= FALSE,													//
		bAlarm4			:= FALSE,													//		
		bAlarm5			:= IN_CmdOpenDC,                                            // Open DC command
		bAlarm6			:= IN_CmdCloseDC,                                           // Close DC Command
		bAlarm7			:= FALSE,                                                   //
		bAlarm8			:= FALSE,                                                   //
		bAlarm9			:= FALSE,                                                   //
		bAlarm10		:= FALSE,                                                   //
		bAlarm11		:= FALSE,                                                   //
		bAlarm12		:= FALSE,                                                   //
		bAlarm13		:= FALSE,                                                   //
		bAlarm14		:= FALSE,                                                   //
		bAlarm15		:= FALSE,                                                   //
		wAlarmCode		=>MesDataExd.MesData.MesEventCode);
END_METHOD

METHOD M_CP
//////////////////
//  Permanent conditions 
/////////////////

VAR 
	// Method local variables (reinitialized at each cycle) 
	
END_VAR


SUPER^.M_CP() ; 




Trig_Cmd_Read(CLK:=IN_CmdToggleRead);
Trig_Cmd_Write(CLK:=IN_CmdToggleWrite);
	
IF Trig_Cmd_Read.Q THEN
	IN_CmdToggleRead := FALSE;
	MesDataExd.MesData.MesCP_Read := NOT MesDataExd.MesData.MesCP_Read;
END_IF


IF Trig_Cmd_Write.Q THEN
	IN_CmdToggleWrite := FALSE;
	MesDataExd.MesData.MesCP_Write := NOT MesDataExd.MesData.MesCP_Write;
END_IF
END_METHOD

METHOD M_Evaluate : BOOL
VAR_INPUT
END_VAR
VAR
	KK : UINT;
	MinVdc : REAL;
	MaxVdc : REAL;
//	MinVdcRackId : UINT;
//	MaxVdcRackId : UINT;
//	MinVdcModuleId : UINT;
//	MaxVdcModuleId : UINT;	
	JJ: INT;
	Temp_Energy: REAL;
END_VAR
 


//Watchdog fixed value :
	AX_DFV[13]
	(
		IN_Addr := ADR(MesDataExd.MesHeartBeat),
		IN_EmptyStruct := ADR(AX_DFV[13]),
		IN_Size := SIZEOF(MesDataExd.MesHeartBeat),
		IN_Duration := ParamTimeWatchdog
	);


MesDataExd.MesUdcMin_RackID := 1 ; 
MesDataExd.MesNbRackNormal := 0 ; 
MesDataExd.MesEconnected := 0;
FOR KK:= 1 TO ParamNbRacks DO 
MesDataExd.AX_Rack[KK].CalRackClosed := MesDataExd.AX_Rack[KK].MesSwitchSensorStatus.2 ; 
	

	FOR JJ:= 1 TO ParamNbRackString DO 
		IF MesDataExd.AX_Rack[KK].AX_RACKSTRING[JJ].MesData.MesUdc = MesDataExd.MesUdcMax THEN MesDataExd.MesUdcMax_RackID := KK ; END_IF  ; 
		IF MesDataExd.AX_Rack[KK].AX_RACKSTRING[JJ].MesData.MesUdc = MesDataExd.MesUdcMin THEN MesDataExd.MesUdcMin_RackID := KK ; END_IF  ; 
		
		IF MesDataExd.AX_Rack[KK].CalRackClosed THEN
		MesDataExd.MesData.MesEconnected  := MesDataExd.MesData.MesEconnected + MesDataExd.AX_Rack[KK].AX_RACKSTRING[JJ].MesData.MesSoH/100 * ParamEnom_Rack ; 
		END_IF
		
	MesDataExd.MesData.MesNbRackNormal := MesDataExd.MesData.MesNbRackNormal + SEL(MesDataExd.AX_Rack[KK].AX_RACKSTRING[JJ].MesAlarm1.6 OR MesDataExd.AX_Rack[KK].AX_RACKSTRING[JJ].MesAlarm1.5 OR MesDataExd.AX_Rack[KK].AX_RACKSTRING[JJ].MesAlarm1.4
										OR MesDataExd.AX_Rack[KK].AX_RACKSTRING[JJ].MesAlarm1.3 OR MesDataExd.AX_Rack[KK].AX_RACKSTRING[JJ].MesAlarm1.2 OR MesDataExd.AX_Rack[KK].AX_RACKSTRING[JJ].MesAlarm1.1
										OR MesDataExd.AX_Rack[KK].AX_RACKSTRING[JJ].MesAlarm1.0 OR MesDataExd.AX_Rack[KK].AX_RACKSTRING[JJ].MesAlarm2.10 OR MesDataExd.AX_Rack[KK].AX_RACKSTRING[JJ].MesAlarm2.9
										OR MesDataExd.AX_Rack[KK].AX_RACKSTRING[JJ].MesAlarm2.8 OR MesDataExd.AX_Rack[KK].AX_RACKSTRING[JJ].MesAlarm2.5 OR MesDataExd.AX_Rack[KK].AX_RACKSTRING[JJ].MesAlarm2.3
										OR MesDataExd.AX_Rack[KK].AX_RACKSTRING[JJ].MesAlarm2.2 OR MesDataExd.AX_Rack[KK].AX_RACKSTRING[JJ].MesAlarm2.1 OR MesDataExd.AX_Rack[KK].AX_RACKSTRING[JJ].MesAlarm3.7
										OR MesDataExd.AX_Rack[KK].AX_RACKSTRING[JJ].MesAlarm3.6 OR MesDataExd.AX_Rack[KK].AX_RACKSTRING[JJ].MesAlarm3.4 OR MesDataExd.AX_Rack[KK].AX_RACKSTRING[JJ].MesAlarm3.2
										OR MesDataExd.AX_Rack[KK].AX_RACKSTRING[JJ].MesAlarm3.1 OR MesDataExd.AX_Rack[KK].AX_RACKSTRING[JJ].MesAlarm3.0 OR MesDataExd.AX_Rack[KK].AX_RACKSTRING[JJ].MesAlarm4.3
										OR MesDataExd.AX_Rack[KK].AX_RACKSTRING[JJ].MesAlarm4.2  OR MesDataExd.AX_Rack[KK].AX_RACKSTRING[JJ].MesAlarm4.1 , 1, 0)* SEL(MesDataExd.AX_Rack[KK].CalRackClosed , 0,1); 
		
	END_FOR
END_FOR
	

// Calculate Econnected value based on calculation if LOC BBMS 
(*IF MesDataExd.MesData.MesComAlarm THEN 
MesDataExd.MesData.CalEconnected := MesDataExd.MesData.CalEconnected + MesDataExd.MesData.CalPdc 
ELSE*)

(*END_IF *)


MesDataExd.MesData.MesPdc	:= MesDataExd.MesData.MesIdc * MesDataExd.MesData.MesUdc / 1000;

Trig_NewDay(clk := CalLocalTimeStruct.wMinute MOD 10 = 0);
Trig_Second(CLK := CalLocalTimeStruct.wMilliseconds < 500);

(*
IF Trig_NewDay.Q THEN
MesDataExd.CalCrateCharge 			:= 0;
MesDataExd.MesData.CalNbPointsDayCharge	:= 0;
	
MesDataExd.MesData.CalCRateDischarge 		:= 0;
MesDataExd.MesData.CalNbPointsDayDischarge	:= 0;
	
MesDataExd.MesData.CalCSoC 				:= 0;
MesDataExd.MesData.CalNbPointsDayCenter	:= 0;
	
MesDataExd.MesData.CalRSoC 				:= 0;
MesDataExd.MesData.CalNbPointsDayRest		:= 0;
END_IF

IF Trig_Second.Q THEN
	IF MesDataExd.MesData.MesPdc < 0 THEN
		E_Throughput_Integrate(IN_DataToIntegrate := MesDataExd.MesData.MesPdc, IN_CmdReset := Trig_NewDay.Q, OUT_IntegrationValue => Temp_Energy);
	MesDataExd.MesData.CalEnergyThroughput := Temp_Energy/3600;
		
	END_IF
	
	IF MesDataExd.MesData.MesSystemMode.14 THEN
	MesDataExd.MesData.CalCrateCharge 				:= MesDataExd.MesData.CalCrateCharge + ABS.MesDataExd.MesData.MesPdc/(ParamEnomRack*ParamNbRacks));
	MesDataExd.MesData.CalNbPointsDayCharge		:= MesDataExd.MesData.CalNbPointsDayCharge + 1;
	END_IF
	
	IF MesDataExd.MesData.MesSystemMode.15 THEN	
	MesDataExd.MesData.CalCRateDischarge 			:= MesDataExd.MesData.CalCRateDischarge + ABS.MesDataExd.MesData.MesPdc/(ParamEnomRack*ParamNbRacks));
	MesDataExd.MesData.CalNbPointsDayDischarge		:= MesDataExd.MesData.CalNbPointsDayDischarge + 1;
	END_IF
	
	IF NOT MesDataExd.MesData.MesSystemMode.14 OR MesDataExd.MesData.MesSystemMode.15) THEN
	MesDataExd.MesData.CalRSoC						:= MesDataExd.MesData.CalRSoC + MesDataExd.MesData.MesSoC;
	MesDataExd.MesData.CalNbPointsDayRest  		:= MesDataExd.MesData.CalNbPointsDayRest + 1;
	END_IF
	
	IF MesDataExd.MesData.MesSystemMode.14 OR MesDataExd.MesData.MesSystemMode.15 THEN
	MesDataExd.MesData.CalCSoC						:= MesDataExd.MesData.CalCSoC + MesDataExd.MesData.MesSoC;
	MesDataExd.MesData.CalNbPointsDayCenter  		:= MesDataExd.MesData.CalNbPointsDayCenter + 1;
	END_IF
END_IF	
*)

SUPER^.M_Evaluate();
END_METHOD

METHOD M_Init
VAR 

END_VAR
MesCP_Read := TRUE;
MesCP_Write := TRUE;
END_METHOD

METHOD M_Read
//////////////////
//  Read CAN 2.0B Variables for racks and BBMS .  
/////////////////

VAR 
	// Method local variables (reinitialized at each cycle) 
	MW 	: FB_MergeWordsToDint ; 

	AX_Addr		: ARRAY[1..2] OF UINT := [16#00	,  16#3E8];
	AX_Qty		: ARRAY[1..3] OF UINT := [	112		, 35	,97	];
	LL			: INT;
	KK			: BYTE;
	CalRackNb	: INT;
	JJ			: BYTE;

END_VAR
// System BMS 
IF  MesDataExd.MesData.MesCP_Read THEN	

	ModbusRead
	(
		pDestAddr 		:= ADR(MesBlock1_Temp),		sIPAddr 		:= ParamIpAddress,			tTimeout 		:= ParamTimeout,
		nTcpPort 		:= ParamTcpPort,				nQuantity 		:= AX_Qty[1],				nMBAddr 		:= AX_Addr[1],				
		cbLength 		:= SIZEOF(MesBlock1_Temp),	nUnitID 		:= ParamUnitID,				ClockRead 		:= Clockread AND  MesDataExd.MesData.MesCP_Read,
		Reset 			:= IN_CmdReset,					ModbusReadAlarm => MesModbusReadAlarm,	ErrorId 		=> MesModbusReadAlarmID
	);



	MesDataExd.MesHeartBeat:=MesBlock1_Temp[0];
	MesDataExd.MesNbRackConnected:=MesBlock1_Temp[1];
	MesDataExd.MesNbRackTot:=MesBlock1_Temp[2];
	MW(WORD_STRONG:= MesBlock1_Temp[ 3], SIGNED:=TRUE, FIX:=0 , SIZE:=1, VAR_OUT := MesDataExd.MesIdcConnected);
	MW(WORD_STRONG:= MesBlock1_Temp[ 4], SIGNED:=FALSE, FIX:=1 , SIZE:=1, VAR_OUT := MesDataExd.MesUdcConnected);
	MW(WORD_STRONG:= MesBlock1_Temp[ 5], SIGNED:=FALSE, FIX:=1 , SIZE:=1, VAR_OUT := MesDataExd.MesUdcConnectedMedian);
	MW(WORD_STRONG:= MesBlock1_Temp[ 6], SIGNED:=FALSE, FIX:=1 , SIZE:=1, VAR_OUT := MesDataExd.MesUdcConnectedMax);
	MW(WORD_STRONG:= MesBlock1_Temp[ 7], SIGNED:=FALSE, FIX:=1 , SIZE:=1, VAR_OUT := MesDataExd.MesUdcConnectedMin);
	MW(WORD_STRONG:= MesBlock1_Temp[ 8], SIGNED:=FALSE, FIX:=1 , SIZE:=1, VAR_OUT := MesDataExd.MesSoCConnected);
	MW(WORD_STRONG:= MesBlock1_Temp[ 9], SIGNED:=FALSE, FIX:=1 , SIZE:=1, VAR_OUT := MesDataExd.MesSoCConnectedMedian);
	MW(WORD_STRONG:= MesBlock1_Temp[ 10], SIGNED:=FALSE, FIX:=1 , SIZE:=1, VAR_OUT := MesDataExd.MesSoCConnectedMax);
	MW(WORD_STRONG:= MesBlock1_Temp[ 11], SIGNED:=FALSE, FIX:=1 , SIZE:=1, VAR_OUT := MesDataExd.MesSoCConnectedMin);
	MW(WORD_STRONG:= MesBlock1_Temp[ 12], SIGNED:=TRUE, FIX:=0 , SIZE:=1, VAR_OUT := MesDataExd.MesData.MesIdc);
	MW(WORD_STRONG:= MesBlock1_Temp[ 13], SIGNED:=FALSE, FIX:=1 , SIZE:=1, VAR_OUT := MesDataExd.MesData.MesUdc);
	MW(WORD_STRONG:= MesBlock1_Temp[ 14], SIGNED:=FALSE, FIX:=1 , SIZE:=1, VAR_OUT := MesDataExd.MesUdcMedian);
	MW(WORD_STRONG:= MesBlock1_Temp[ 15], SIGNED:=FALSE, FIX:=1 , SIZE:=1, VAR_OUT := MesDataExd.MesUdcMax);
	MW(WORD_STRONG:= MesBlock1_Temp[ 16], SIGNED:=FALSE, FIX:=1 , SIZE:=1, VAR_OUT := MesDataExd.MesUdcMin);
	MW(WORD_STRONG:= MesBlock1_Temp[ 17], SIGNED:=FALSE, FIX:=1 , SIZE:=1, VAR_OUT := MesDataExd.MesData.MesSoC);
	MW(WORD_STRONG:= MesBlock1_Temp[ 18], SIGNED:=FALSE, FIX:=1 , SIZE:=1, VAR_OUT := MesDataExd.MesSoCMedian);
	MW(WORD_STRONG:= MesBlock1_Temp[ 19], SIGNED:=FALSE, FIX:=1 , SIZE:=1, VAR_OUT := MesDataExd.MesSoCMax);
	MW(WORD_STRONG:= MesBlock1_Temp[ 20], SIGNED:=FALSE, FIX:=1 , SIZE:=1, VAR_OUT := MesDataExd.MesSoCMin);
	MW(WORD_STRONG:= MesBlock1_Temp[ 21], SIGNED:=FALSE, FIX:=1 , SIZE:=1, VAR_OUT := MesDataExd.MesData.MesSoH);
	MW(WORD_STRONG:= MesBlock1_Temp[ 22], SIGNED:=FALSE, FIX:=1 , SIZE:=1, VAR_OUT := MesDataExd.MesSoHMedian);
	MW(WORD_STRONG:= MesBlock1_Temp[ 23], SIGNED:=FALSE, FIX:=1 , SIZE:=1, VAR_OUT := MesDataExd.MesSoHMax);
	MW(WORD_STRONG:= MesBlock1_Temp[ 24], SIGNED:=FALSE, FIX:=1 , SIZE:=1, VAR_OUT := MesDataExd.MesSoHMin);
	MW(WORD_STRONG:= MesBlock1_Temp[ 25], SIGNED:=FALSE, FIX:=3 , SIZE:=1, VAR_OUT := MesDataExd.MesUdc_Cell);
	MW(WORD_STRONG:= MesBlock1_Temp[ 26], SIGNED:=FALSE, FIX:=3 , SIZE:=1, VAR_OUT := MesDataExd.MesUdcMedian_Cell);
	MW(WORD_STRONG:= MesBlock1_Temp[ 27], SIGNED:=FALSE, FIX:=3 , SIZE:=1, VAR_OUT := MesDataExd.MesUdcMax_Cell);
	MesDataExd.MesUdcMax_Cell_RackID:=MesBlock1_Temp[28];
	MW(WORD_STRONG:= MesBlock1_Temp[ 29], SIGNED:=FALSE, FIX:=3 , SIZE:=1, VAR_OUT := MesDataExd.MesUdcMin_Cell);
	MesDataExd.MesUdcMin_Cell_RackID:=MesBlock1_Temp[30];
	MW(WORD_STRONG:= MesBlock1_Temp[ 31], SIGNED:=FALSE, FIX:=3 , SIZE:=1, VAR_OUT := MesDataExd.MesUdcDiffMax_Cell);
	MesDataExd.MesUdcDiffMax_Cell_RackID:=MesBlock1_Temp[32];
	MW(WORD_STRONG:= MesBlock1_Temp[ 33], SIGNED:=TRUE, FIX:=2 , SIZE:=1, VAR_OUT := MesDataExd.MesTmp_Cell);
	MW(WORD_STRONG:= MesBlock1_Temp[ 34], SIGNED:=TRUE, FIX:=2 , SIZE:=1, VAR_OUT := MesDataExd.MesTmpMedian_Cell);
	MW(WORD_STRONG:= MesBlock1_Temp[ 35], SIGNED:=TRUE, FIX:=2 , SIZE:=1, VAR_OUT := MesDataExd.MesTmpMax_Cell);
	MesDataExd.MesTmpMax_Cell_RackID:=MesBlock1_Temp[36];
	MW(WORD_STRONG:= MesBlock1_Temp[ 37], SIGNED:=TRUE, FIX:=2 , SIZE:=1, VAR_OUT := MesDataExd.MesTmpMin_Cell);
	MesDataExd.MesTmpMin_Cell_RackID:=MesBlock1_Temp[38];
	MW(WORD_STRONG:= MesBlock1_Temp[ 39], SIGNED:=FALSE, FIX:=2 , SIZE:=1, VAR_OUT := MesDataExd.MesTmpDiffMax_Cell);
	MesDataExd.MesTmpDiffMax_Cell_RackID:=MesBlock1_Temp[40];
	MW(WORD_STRONG:= MesBlock1_Temp[ 41], Word_WEAK:= MesBlock1_Temp[42], SIGNED:=FALSE, FIX:=1 , SIZE:=2, VAR_OUT := MesDataExd.MesData.MesCCL);
	MW(WORD_STRONG:= MesBlock1_Temp[ 43], Word_WEAK:= MesBlock1_Temp[44], SIGNED:=FALSE, FIX:=1 , SIZE:=2, VAR_OUT := MesDataExd.MesData.MesDCL);
	MW(WORD_STRONG:= MesBlock1_Temp[ 45], Word_WEAK:= MesBlock1_Temp[46], SIGNED:=FALSE, FIX:=2 , SIZE:=2, VAR_OUT := MesDataExd.MesData.MesCPL);
	MW(WORD_STRONG:= MesBlock1_Temp[ 47], Word_WEAK:= MesBlock1_Temp[48], SIGNED:=FALSE, FIX:=2 , SIZE:=2, VAR_OUT := MesDataExd.MesData.MesDPL);
	
	MesDataExd.MesData.MesECharge :=  LREAL_TO_REAL(LWORD_TO_LREAL(SHL(WORD_TO_LWORD(MesBlock1_Temp[ 49]),48) OR SHL(WORD_TO_LWORD(MesBlock1_Temp[ 50]),32) OR SHL(WORD_TO_LWORD(MesBlock1_Temp[ 51]),16) OR WORD_TO_LWORD(MesBlock1_Temp[ 52]))/ EXPT(10,3) ); 
	MesDataExd.MesData.MesEDischarge :=   LREAL_TO_REAL(LWORD_TO_LREAL(SHL(WORD_TO_LWORD(MesBlock1_Temp[ 53]),48) OR SHL(WORD_TO_LWORD(MesBlock1_Temp[ 54]),32) OR SHL(WORD_TO_LWORD(MesBlock1_Temp[ 55]),16) OR WORD_TO_LWORD(MesBlock1_Temp[ 56]))/ EXPT(10,3)) ; 
	
	MesDataExd.MesWatchdog:=MesBlock1_Temp[57];
	MW(WORD_STRONG:= MesBlock1_Temp[ 58], SIGNED:=FALSE, FIX:=1 , SIZE:=1, VAR_OUT := MesDataExd.MesUdc_PartialOp);
	MesDataExd.MesUdc_PartialOp_RackID:=MesBlock1_Temp[59];
	MesDataExd.MesUdc_PartialOp_StringID:=MesBlock1_Temp[60];
	MesDataExd.MesSystemCommandStatus:=MesBlock1_Temp[71];
	MesDataExd.MesSystemMode:=MesBlock1_Temp[72];
	MesDataExd.MesSystemMode2:=MesBlock1_Temp[73];
	MesDataExd.MesAlarm1:=MesBlock1_Temp[74];
	MesDataExd.MesAlarm2:=MesBlock1_Temp[75];
	MesDataExd.MesRackAlarm1:=MesBlock1_Temp[76];
	MesDataExd.MesRackAlarm2:=MesBlock1_Temp[77];
	MesDataExd.MesRackProtection1:=MesBlock1_Temp[78];
	MesDataExd.MesRackProtection2:=MesBlock1_Temp[79];
	MesDataExd.MesRackStringAlarm1:=MesBlock1_Temp[80];
	MesDataExd.MesRackStringAlarm2:=MesBlock1_Temp[81];
	MesDataExd.MesRackStringAlarm3:=MesBlock1_Temp[82];
	MesDataExd.MesRackStringAlarm4:=MesBlock1_Temp[83];
	MesDataExd.MesRackStringProtection1:=MesBlock1_Temp[84];
	MesDataExd.MesRackStringProtection2:=MesBlock1_Temp[85];
	MesDataExd.MesRackStringProtection3:=MesBlock1_Temp[86];
	MesDataExd.MesRackStringProtection4:=MesBlock1_Temp[87];
	MesDataExd.MesDiStatus:=MesBlock1_Temp[88];
	MesDataExd.MesDoStatus:=MesBlock1_Temp[89];
	MesDataExd.MesSystemConfig1:=MesBlock1_Temp[90];
	MesDataExd.MesSystemConfig2:=MesBlock1_Temp[91];
	MesDataExd.MesRackStringState:=MesBlock1_Temp[92];
	MesDataExd.MesData.ParamNbRacks:=MesBlock1_Temp[105];
	MesDataExd.MesData.ParamNbModule:=MesBlock1_Temp[106];
	MesDataExd.MesData.ParamStringNbMin:=MesBlock1_Temp[107];
	MW(WORD_STRONG:= MesBlock1_Temp[ 108], SIGNED:=FALSE, FIX:=0 , SIZE:=1, VAR_OUT := MesDataExd.MesData.ParamUdiff);
END_IF

// RACKS 

// READ TCU DATA 
CTU_ClockRead(CU:=ClockRead , PV:= REAL_TO_WORD(ParamNbRacks/(ParamNbReadAtOnce))+1 ) ; 
CTU_ClockRead(RESET:= CTU_ClockRead.Q ) ; 
LL:= (CTU_ClockRead.CV)  ; // At every Clock Read , we read 10 new racks We reset once all trackers have been read.  


TON_ClockRead(IN:= ClockRead , PT:= ParamClockReadRack_Delay  ) ; // Allow to leave 200ms between the system data read and the racks reading . 

//RACK 
FOR KK:= 1 TO ParamNbReadAtOnce DO 
	
	CalRackNb := LL*ParamNbReadAtOnce+KK; 	
	IF CalRackNb > ParamNbRacks THEN 
		EXIT ; 
	END_IF	
	
	IF MesDataExd.MesData.MesCP_Read THEN
		ModbusReadrack[(ParamNbRackString+1)*(KK-1)+1]
			(
			pDestAddr 		:= ADR(MesBlock2_Temp[(ParamNbRackString+1)*(KK-1)+1]),		
			sIPAddr 		:= ParamIpAddress,			
			tTimeout 		:= ParamTimeout,
			nTcpPort 		:= ParamTcpPort,				
			nQuantity 		:= AX_Qty[2],				
			nMBAddr 		:= AX_Addr[2] + (CalRackNb-1)*360,				
			cbLength 		:= SIZEOF(MesBlock2_Temp[(ParamNbRackString+1)*(KK-1)+1]),	
			nUnitID 		:= ParamUnitID,				
			ClockRead 		:= TON_ClockRead.Q AND MesDataExd.MesData.MesCP_Read,
			Reset 			:= IN_CmdReset,					
			ModbusReadAlarm => MesModbusReadAlarm2[(ParamNbRackString+1)*(KK-1)+1],	
			ErrorId 		=> MesModbusReadAlarmID2[(ParamNbRackString+1)*(KK-1)+1]
		);
	

	// DATA
		IF ModbusReadrack[(ParamNbRackString+1)*(KK-1)+1].OUT_Completed THEN 
		MesDataExd.AX_Rack[CalRackNb].ParamNbStrings:=MesBlock2_Temp[(ParamNbRackString+1)*(KK-1)+1][0];
		MesDataExd.AX_Rack[CalRackNb].MesHeartBeat:=MesBlock2_Temp[(ParamNbRackString+1)*(KK-1)+1][1];
		MesDataExd.AX_Rack[CalRackNb].MesAlarm1:=MesBlock2_Temp[(ParamNbRackString+1)*(KK-1)+1][2];
		MesDataExd.AX_Rack[CalRackNb].MesAlarm2:=MesBlock2_Temp[(ParamNbRackString+1)*(KK-1)+1][3];
		MesDataExd.AX_Rack[CalRackNb].MesProtection1:=MesBlock2_Temp[(ParamNbRackString+1)*(KK-1)+1][4];
		MesDataExd.AX_Rack[CalRackNb].MesProtection2:=MesBlock2_Temp[(ParamNbRackString+1)*(KK-1)+1][5];
		MesDataExd.AX_Rack[CalRackNb].MesSwitchControlStatus:=MesBlock2_Temp[(ParamNbRackString+1)*(KK-1)+1][6];
		MesDataExd.AX_Rack[CalRackNb].MesSwitchSensorStatus:=MesBlock2_Temp[(ParamNbRackString+1)*(KK-1)+1][7];
			MW(WORD_STRONG:= MesBlock2_Temp[(ParamNbRackString+1)*(KK-1)+1][ 10], 	SIGNED:=FALSE, FIX:=1 , SIZE:=1, VAR_OUT := MesDataExd.AX_Rack[CalRackNb].MesUSwtchGrPackPlus);
			MW(WORD_STRONG:= MesBlock2_Temp[(ParamNbRackString+1)*(KK-1)+1][ 12], 	SIGNED:=TRUE, FIX:=0 , SIZE:=1, VAR_OUT := MesDataExd.AX_Rack[CalRackNb].MesTempPCB);
		MesDataExd.AX_Rack[CalRackNb].MesIdcFaultLvl:=MesBlock2_Temp[(ParamNbRackString+1)*(KK-1)+1][23];
		MesDataExd.AX_Rack[CalRackNb].MesDcOpenCount:=MesBlock2_Temp[(ParamNbRackString+1)*(KK-1)+1][24];
		MesDataExd.AX_Rack[CalRackNb].MesDcCloseCount:=MesBlock2_Temp[(ParamNbRackString+1)*(KK-1)+1][25];
		END_IF
	END_IF
	// RACK STRING 
	FOR JJ:= 1 TO ParamNbRackString DO 
		IF MesDataExd.MesData.MesCP_Read THEN	
			ModbusReadrack[(ParamNbRackString+1)*(KK-1)+JJ+1]
				(
				pDestAddr 		:= ADR(MesBlock2_Temp[(ParamNbRackString+1)*(KK-1)+JJ+1]),		
				sIPAddr 		:= ParamIpAddress,			
				tTimeout 		:= ParamTimeout,
				nTcpPort 		:= ParamTcpPort,				
				nQuantity 		:= AX_Qty[3],				
				nMBAddr 		:= AX_Addr[2] + (CalRackNb-1)*360 + JJ*120,				
				cbLength 		:= SIZEOF(MesBlock2_Temp[(ParamNbRackString+1)*(KK-1)+JJ+1]),	
				nUnitID 		:= ParamUnitID,				
				ClockRead 		:= TON_ClockRead.Q AND MesDataExd.MesData.MesCP_Read,
				Reset 			:= IN_CmdReset,					
				ModbusReadAlarm => MesModbusReadAlarm2[(ParamNbRackString+1)*(KK-1)+JJ+1],	
				ErrorId 		=> MesModbusReadAlarmID2[(ParamNbRackString+1)*(KK-1)+JJ+1]
			);

		//DATA
			IF ModbusReadrack[(ParamNbRackString+1)*(KK-1)+JJ+1].OUT_Completed THEN 
			MesDataExd.AX_RACK[CalrackNb].AX_RACKSTRING[JJ].MesMode:=MesBlock2_Temp[(ParamNbRackString+1)*(KK-1)+JJ+1][0];
			MesDataExd.AX_RACK[CalrackNb].AX_RACKSTRING[JJ].MesAlarm1:=MesBlock2_Temp[(ParamNbRackString+1)*(KK-1)+JJ+1][2];
			MesDataExd.AX_RACK[CalrackNb].AX_RACKSTRING[JJ].MesAlarm2:=MesBlock2_Temp[(ParamNbRackString+1)*(KK-1)+JJ+1][3];
			MesDataExd.AX_RACK[CalrackNb].AX_RACKSTRING[JJ].MesAlarm3:=MesBlock2_Temp[(ParamNbRackString+1)*(KK-1)+JJ+1][4];
			MesDataExd.AX_RACK[CalrackNb].AX_RACKSTRING[JJ].MesAlarm4:=MesBlock2_Temp[(ParamNbRackString+1)*(KK-1)+JJ+1][5];
			MesDataExd.AX_RACK[CalrackNb].AX_RACKSTRING[JJ].MesProtection1:=MesBlock2_Temp[(ParamNbRackString+1)*(KK-1)+JJ+1][6];
			MesDataExd.AX_RACK[CalrackNb].AX_RACKSTRING[JJ].MesProtection2:=MesBlock2_Temp[(ParamNbRackString+1)*(KK-1)+JJ+1][7];
			MesDataExd.AX_RACK[CalrackNb].AX_RACKSTRING[JJ].MesProtection3:=MesBlock2_Temp[(ParamNbRackString+1)*(KK-1)+JJ+1][8];
			MesDataExd.AX_RACK[CalrackNb].AX_RACKSTRING[JJ].MesProtection4:=MesBlock2_Temp[(ParamNbRackString+1)*(KK-1)+JJ+1][9];
			MesDataExd.AX_RACK[CalrackNb].AX_RACKSTRING[JJ].MesControlStatus:=MesBlock2_Temp[(ParamNbRackString+1)*(KK-1)+JJ+1][10];
				MW(WORD_STRONG:= MesBlock2_Temp[(ParamNbRackString+1)*(KK-1)+JJ+1][ 13], SIGNED:=FALSE, FIX:=1 , SIZE:=1, VAR_OUT := MesDataExd.AX_RACK[CalrackNb].AX_RACKSTRING[JJ].MesData.MesUdc);
				MW(WORD_STRONG:= MesBlock2_Temp[(ParamNbRackString+1)*(KK-1)+JJ+1][ 14], SIGNED:=FALSE, FIX:=1 , SIZE:=1, VAR_OUT := MesDataExd.AX_RACK[CalrackNb].AX_RACKSTRING[JJ].MesUdc_ModuleSum);
				MW(WORD_STRONG:= MesBlock2_Temp[(ParamNbRackString+1)*(KK-1)+JJ+1][ 15], SIGNED:=FALSE, FIX:=1 , SIZE:=1, VAR_OUT := MesDataExd.AX_RACK[CalrackNb].AX_RACKSTRING[JJ].MesUdc_CellSum);
				MW(WORD_STRONG:= MesBlock2_Temp[(ParamNbRackString+1)*(KK-1)+JJ+1][ 16], SIGNED:=TRUE, FIX:=1 , SIZE:=1, VAR_OUT := MesDataExd.AX_RACK[CalrackNb].AX_RACKSTRING[JJ].MesData.MesIdc);
				MW(WORD_STRONG:= MesBlock2_Temp[(ParamNbRackString+1)*(KK-1)+JJ+1][ 17], SIGNED:=TRUE, FIX:=1 , SIZE:=1, VAR_OUT := MesDataExd.AX_RACK[CalrackNb].AX_RACKSTRING[JJ].MesIdc_Avg);
				MW(WORD_STRONG:= MesBlock2_Temp[(ParamNbRackString+1)*(KK-1)+JJ+1][ 18], SIGNED:=FALSE, FIX:=1 , SIZE:=1, VAR_OUT := MesDataExd.AX_RACK[CalrackNb].AX_RACKSTRING[JJ].MesData.MesSoC);
				MW(WORD_STRONG:= MesBlock2_Temp[(ParamNbRackString+1)*(KK-1)+JJ+1][ 19], SIGNED:=FALSE, FIX:=1 , SIZE:=1, VAR_OUT := MesDataExd.AX_RACK[CalrackNb].AX_RACKSTRING[JJ].MesData.MesSoH);
				MW(WORD_STRONG:= MesBlock2_Temp[(ParamNbRackString+1)*(KK-1)+JJ+1][ 20], SIGNED:=FALSE, FIX:=1 , SIZE:=1, VAR_OUT := MesDataExd.AX_RACK[CalrackNb].AX_RACKSTRING[JJ].MesCCL);
				MW(WORD_STRONG:= MesBlock2_Temp[(ParamNbRackString+1)*(KK-1)+JJ+1][ 21], SIGNED:=FALSE, FIX:=1 , SIZE:=1, VAR_OUT := MesDataExd.AX_RACK[CalrackNb].AX_RACKSTRING[JJ].MesDCL);
				MW(WORD_STRONG:= MesBlock2_Temp[(ParamNbRackString+1)*(KK-1)+JJ+1][ 22], SIGNED:=FALSE, FIX:=2 , SIZE:=1, VAR_OUT := MesDataExd.AX_RACK[CalrackNb].AX_RACKSTRING[JJ].MesCPL);
				MW(WORD_STRONG:= MesBlock2_Temp[(ParamNbRackString+1)*(KK-1)+JJ+1][ 23], SIGNED:=FALSE, FIX:=2 , SIZE:=1, VAR_OUT := MesDataExd.AX_RACK[CalrackNb].AX_RACKSTRING[JJ].MesDPL);
				
			MesDataExd.AX_RACK[CalrackNb].AX_RACKSTRING[JJ].MesECharge := LREAL_TO_REAL(LWORD_TO_LREAL(SHL(WORD_TO_LWORD(MesBlock2_Temp[(ParamNbRackString+1)*(KK-1)+JJ+1][ 24]),48) OR SHL(WORD_TO_LWORD(MesBlock2_Temp[(ParamNbRackString+1)*(KK-1)+JJ+1][ 25]),32) OR SHL(WORD_TO_LWORD(MesBlock2_Temp[(ParamNbRackString+1)*(KK-1)+JJ+1][ 26]),16) OR WORD_TO_LWORD(MesBlock2_Temp[(ParamNbRackString+1)*(KK-1)+JJ+1][ 27]))/ EXPT(10,3) ); 
				
			MesDataExd.AX_RACK[CalrackNb].AX_RACKSTRING[JJ].MesEDischarge := LREAL_TO_REAL(LWORD_TO_LREAL(SHL(WORD_TO_LWORD(MesBlock2_Temp[(ParamNbRackString+1)*(KK-1)+JJ+1][ 28]),48) OR SHL(WORD_TO_LWORD(MesBlock2_Temp[(ParamNbRackString+1)*(KK-1)+JJ+1][ 29]),32) OR SHL(WORD_TO_LWORD(MesBlock2_Temp[(ParamNbRackString+1)*(KK-1)+JJ+1][ 30]),16) OR WORD_TO_LWORD(MesBlock2_Temp[(ParamNbRackString+1)*(KK-1)+JJ+1][ 31]))/ EXPT(10,3) ); 
				
			MesDataExd.AX_RACK[CalrackNb].AX_RACKSTRING[JJ].MesOff_ModuleID:=MesBlock2_Temp[(ParamNbRackString+1)*(KK-1)+JJ+1][36];
			MesDataExd.AX_RACK[CalrackNb].AX_RACKSTRING[JJ].MesComError_ModuleID:=MesBlock2_Temp[(ParamNbRackString+1)*(KK-1)+JJ+1][37];
				MW(WORD_STRONG:= MesBlock2_Temp[(ParamNbRackString+1)*(KK-1)+JJ+1][ 38], SIGNED:=FALSE, FIX:=3 , SIZE:=1, VAR_OUT := MesDataExd.AX_RACK[CalrackNb].AX_RACKSTRING[JJ].MesUdcDiffMax_Cell);
				MW(WORD_STRONG:= MesBlock2_Temp[(ParamNbRackString+1)*(KK-1)+JJ+1][ 39], SIGNED:=FALSE, FIX:=3 , SIZE:=1, VAR_OUT := MesDataExd.AX_RACK[CalrackNb].AX_RACKSTRING[JJ].MesData.MesUdc_Cell);
				MW(WORD_STRONG:= MesBlock2_Temp[(ParamNbRackString+1)*(KK-1)+JJ+1][ 40], SIGNED:=FALSE, FIX:=3 , SIZE:=1, VAR_OUT := MesDataExd.AX_RACK[CalrackNb].AX_RACKSTRING[JJ].MesData.MesUdcMax_Cell);
			MesDataExd.AX_RACK[CalrackNb].AX_RACKSTRING[JJ].MesData.MesIDModule_UdcMax_Cell:=MesBlock2_Temp[(ParamNbRackString+1)*(KK-1)+JJ+1][41];
			MesDataExd.AX_RACK[CalrackNb].AX_RACKSTRING[JJ].MesUdcMax1_Cell_CellID:=MesBlock2_Temp[(ParamNbRackString+1)*(KK-1)+JJ+1][42];
				MW(WORD_STRONG:= MesBlock2_Temp[(ParamNbRackString+1)*(KK-1)+JJ+1][ 43], SIGNED:=FALSE, FIX:=3 , SIZE:=1, VAR_OUT := MesDataExd.AX_RACK[CalrackNb].AX_RACKSTRING[JJ].MesData.MesUdcMin_Cell);
			MesDataExd.AX_RACK[CalrackNb].AX_RACKSTRING[JJ].MesData.MesIDModule_UdcMin_Cell:=MesBlock2_Temp[(ParamNbRackString+1)*(KK-1)+JJ+1][44];
			MesDataExd.AX_RACK[CalrackNb].AX_RACKSTRING[JJ].MesUdcMin1_Cell_CellID:=MesBlock2_Temp[(ParamNbRackString+1)*(KK-1)+JJ+1][45];
				MW(WORD_STRONG:= MesBlock2_Temp[(ParamNbRackString+1)*(KK-1)+JJ+1][ 46], SIGNED:=FALSE, FIX:=3 , SIZE:=1, VAR_OUT := MesDataExd.AX_RACK[CalrackNb].AX_RACKSTRING[JJ].MesUdcMax2_Cell);
			MesDataExd.AX_RACK[CalrackNb].AX_RACKSTRING[JJ].MesUdcMax2_Cell_ModuleID:=MesBlock2_Temp[(ParamNbRackString+1)*(KK-1)+JJ+1][47];
			MesDataExd.AX_RACK[CalrackNb].AX_RACKSTRING[JJ].MesUdcMax2_Cell_CellID:=MesBlock2_Temp[(ParamNbRackString+1)*(KK-1)+JJ+1][48];
				MW(WORD_STRONG:= MesBlock2_Temp[(ParamNbRackString+1)*(KK-1)+JJ+1][ 49], SIGNED:=FALSE, FIX:=3 , SIZE:=1, VAR_OUT := MesDataExd.AX_RACK[CalrackNb].AX_RACKSTRING[JJ].MesUdcMin2_Cell);
			MesDataExd.AX_RACK[CalrackNb].AX_RACKSTRING[JJ].MesUdcMin2_Cell_ModuleID:=MesBlock2_Temp[(ParamNbRackString+1)*(KK-1)+JJ+1][50];
			MesDataExd.AX_RACK[CalrackNb].AX_RACKSTRING[JJ].MesUdcMin2_Cell_CellID:=MesBlock2_Temp[(ParamNbRackString+1)*(KK-1)+JJ+1][51];
				MW(WORD_STRONG:= MesBlock2_Temp[(ParamNbRackString+1)*(KK-1)+JJ+1][ 52], SIGNED:=FALSE, FIX:=2 , SIZE:=1, VAR_OUT := MesDataExd.AX_RACK[CalrackNb].AX_RACKSTRING[JJ].MesTempDiffMax_Cell);
				MW(WORD_STRONG:= MesBlock2_Temp[(ParamNbRackString+1)*(KK-1)+JJ+1][ 53], SIGNED:=TRUE, FIX:=2 , SIZE:=1, VAR_OUT := MesDataExd.AX_RACK[CalrackNb].AX_RACKSTRING[JJ].MesTemp_Cell);
				MW(WORD_STRONG:= MesBlock2_Temp[(ParamNbRackString+1)*(KK-1)+JJ+1][ 54], SIGNED:=TRUE, FIX:=2 , SIZE:=1, VAR_OUT := MesDataExd.AX_RACK[CalrackNb].AX_RACKSTRING[JJ].MesTempMax1_Cell);
			MesDataExd.AX_RACK[CalrackNb].AX_RACKSTRING[JJ].MesTempMax1_Cell_ModuleID:=MesBlock2_Temp[(ParamNbRackString+1)*(KK-1)+JJ+1][55];
			MesDataExd.AX_RACK[CalrackNb].AX_RACKSTRING[JJ].MesTempMax1_Cell_CellID:=MesBlock2_Temp[(ParamNbRackString+1)*(KK-1)+JJ+1][56];
				MW(WORD_STRONG:= MesBlock2_Temp[(ParamNbRackString+1)*(KK-1)+JJ+1][ 57], SIGNED:=TRUE, FIX:=2 , SIZE:=1, VAR_OUT := MesDataExd.AX_RACK[CalrackNb].AX_RACKSTRING[JJ].MesTempMin1_Cell);
			MesDataExd.AX_RACK[CalrackNb].AX_RACKSTRING[JJ].MesTempMin1_Cell_ModuleID:=MesBlock2_Temp[(ParamNbRackString+1)*(KK-1)+JJ+1][58];
			MesDataExd.AX_RACK[CalrackNb].AX_RACKSTRING[JJ].MesTempMin1_Cell_CellID:=MesBlock2_Temp[(ParamNbRackString+1)*(KK-1)+JJ+1][59];
				MW(WORD_STRONG:= MesBlock2_Temp[(ParamNbRackString+1)*(KK-1)+JJ+1][ 60], SIGNED:=TRUE, FIX:=2 , SIZE:=1, VAR_OUT := MesDataExd.AX_RACK[CalrackNb].AX_RACKSTRING[JJ].MesTempMax2_Cell);
			MesDataExd.AX_RACK[CalrackNb].AX_RACKSTRING[JJ].MesTempMax2_Cell_ModuleID:=MesBlock2_Temp[(ParamNbRackString+1)*(KK-1)+JJ+1][61];
			MesDataExd.AX_RACK[CalrackNb].AX_RACKSTRING[JJ].MesTempMax2_Cell_CellID:=MesBlock2_Temp[(ParamNbRackString+1)*(KK-1)+JJ+1][62];
				MW(WORD_STRONG:= MesBlock2_Temp[(ParamNbRackString+1)*(KK-1)+JJ+1][ 63], SIGNED:=TRUE, FIX:=2 , SIZE:=1, VAR_OUT := MesDataExd.AX_RACK[CalrackNb].AX_RACKSTRING[JJ].MesTempMin2_Cell);
			MesDataExd.AX_RACK[CalrackNb].AX_RACKSTRING[JJ].MesTempMin2_Cell_ModuleID:=MesBlock2_Temp[(ParamNbRackString+1)*(KK-1)+JJ+1][64];
			MesDataExd.AX_RACK[CalrackNb].AX_RACKSTRING[JJ].MesTempMin2_Cell_CellID:=MesBlock2_Temp[(ParamNbRackString+1)*(KK-1)+JJ+1][65];
				MW(WORD_STRONG:= MesBlock2_Temp[(ParamNbRackString+1)*(KK-1)+JJ+1][ 66], SIGNED:=TRUE, FIX:=2 , SIZE:=1, VAR_OUT := MesDataExd.AX_RACK[CalrackNb].AX_RACKSTRING[JJ].MesTempPCBMax);
			MesDataExd.AX_RACK[CalrackNb].AX_RACKSTRING[JJ].MesTempPCBMax_ModuleID:=MesBlock2_Temp[(ParamNbRackString+1)*(KK-1)+JJ+1][67];
				MW(WORD_STRONG:= MesBlock2_Temp[(ParamNbRackString+1)*(KK-1)+JJ+1][ 68], SIGNED:=TRUE, FIX:=2 , SIZE:=1, VAR_OUT := MesDataExd.AX_RACK[CalrackNb].AX_RACKSTRING[JJ].MesTempPCBMin);
			MesDataExd.AX_RACK[CalrackNb].AX_RACKSTRING[JJ].MesTempPCBMin_ModuleID:=MesBlock2_Temp[(ParamNbRackString+1)*(KK-1)+JJ+1][69];
			MesDataExd.AX_RACK[CalrackNb].AX_RACKSTRING[JJ].MesSensorStatus:=MesBlock2_Temp[(ParamNbRackString+1)*(KK-1)+JJ+1][75];
			MesDataExd.AX_RACK[CalrackNb].AX_RACKSTRING[JJ].MesModuleScanStatus:=MesBlock2_Temp[(ParamNbRackString+1)*(KK-1)+JJ+1][76];
			MesDataExd.AX_RACK[CalrackNb].AX_RACKSTRING[JJ].MesModuleBalancingStatus:=MesBlock2_Temp[(ParamNbRackString+1)*(KK-1)+JJ+1][77];
			MesDataExd.AX_RACK[CalrackNb].AX_RACKSTRING[JJ].MesModuleAddressStatus:=MesBlock2_Temp[(ParamNbRackString+1)*(KK-1)+JJ+1][78];
			MesDataExd.AX_RACK[CalrackNb].AX_RACKSTRING[JJ].MesModuleVoltageStatus:=MesBlock2_Temp[(ParamNbRackString+1)*(KK-1)+JJ+1][79];
			MesDataExd.AX_RACK[CalrackNb].AX_RACKSTRING[JJ].MesModuleTemperatureStatus:=MesBlock2_Temp[(ParamNbRackString+1)*(KK-1)+JJ+1][80];
			MesDataExd.AX_RACK[CalrackNb].AX_RACKSTRING[JJ].MesData.MesIDState:=MesBlock2_Temp[(ParamNbRackString+1)*(KK-1)+JJ+1][87];
				
				MW(WORD_STRONG:= MesBlock2_Temp[(ParamNbRackString+1)*(KK-1)+JJ+1][ 81], 	SIGNED:=FALSE, FIX:=2 , SIZE:=1, VAR_OUT := MesDataExd.AX_RACK[CalrackNb].AX_RACKSTRING[JJ].MesUdcDiffCellMax);
				MW(WORD_STRONG:= MesBlock2_Temp[(ParamNbRackString+1)*(KK-1)+JJ+1][ 82], 	SIGNED:=FALSE, FIX:=2 , SIZE:=1, VAR_OUT := MesDataExd.AX_RACK[CalrackNb].AX_RACKSTRING[JJ].MesUdcDiffModuleMax);
			MesDataExd.AX_RACK[CalrackNb].AX_RACKSTRING[JJ].MesUdcDiffModuleMax_ModuleID:=MesBlock2_Temp[(ParamNbRackString+1)*(KK-1)+JJ+1][83];
				MW(WORD_STRONG:= MesBlock2_Temp[(ParamNbRackString+1)*(KK-1)+JJ+1][ 84], 	SIGNED:=FALSE, FIX:=2 , SIZE:=1, VAR_OUT := MesDataExd.AX_RACK[CalrackNb].AX_RACKSTRING[JJ].MesUdcDiffCellMin);
				MW(WORD_STRONG:= MesBlock2_Temp[(ParamNbRackString+1)*(KK-1)+JJ+1][ 85], 	SIGNED:=FALSE, FIX:=2 , SIZE:=1, VAR_OUT := MesDataExd.AX_RACK[CalrackNb].AX_RACKSTRING[JJ].MesUdcDiffModuleMin);
			MesDataExd.AX_RACK[CalrackNb].AX_RACKSTRING[JJ].MesUdcDiffModuleMin_ModuleID:=MesBlock2_Temp[(ParamNbRackString+1)*(KK-1)+JJ+1][86]	;
				MW(WORD_STRONG:= MesBlock2_Temp[(ParamNbRackString+1)*(KK-1)+JJ+1][ 88], 	SIGNED:=FALSE, FIX:=0 , SIZE:=1, VAR_OUT := MesDataExd.AX_RACK[CalrackNb].AX_RACKSTRING[JJ].MesCellVDist_under20mV);
				MW(WORD_STRONG:= MesBlock2_Temp[(ParamNbRackString+1)*(KK-1)+JJ+1][ 89], 	SIGNED:=FALSE, FIX:=0 , SIZE:=1, VAR_OUT := MesDataExd.AX_RACK[CalrackNb].AX_RACKSTRING[JJ].MesCellVDist_underVimbAlarm );
				MW(WORD_STRONG:= MesBlock2_Temp[(ParamNbRackString+1)*(KK-1)+JJ+1][ 90], 	SIGNED:=FALSE, FIX:=0 , SIZE:=1, VAR_OUT := MesDataExd.AX_RACK[CalrackNb].AX_RACKSTRING[JJ].MesCellVDist_underVimbProtection );
				MW(WORD_STRONG:= MesBlock2_Temp[(ParamNbRackString+1)*(KK-1)+JJ+1][ 91], 	SIGNED:=FALSE, FIX:=0 , SIZE:=1, VAR_OUT := MesDataExd.AX_RACK[CalrackNb].AX_RACKSTRING[JJ].MesCellVDist_VimbProtection );
			MesDataExd.AX_RACK[CalrackNb].AX_RACKSTRING[JJ].MesCellBalancingCntMax:=MesBlock2_Temp[(ParamNbRackString+1)*(KK-1)+JJ+1][92];
			MesDataExd.AX_RACK[CalrackNb].AX_RACKSTRING[JJ].MesCellBalancingCntMax_ModuleID:=MesBlock2_Temp[(ParamNbRackString+1)*(KK-1)+JJ+1][93];
			MesDataExd.AX_RACK[CalrackNb].AX_RACKSTRING[JJ].MesCellBalancingCntMax_CellID:=MesBlock2_Temp[(ParamNbRackString+1)*(KK-1)+JJ+1][94];
				MW(WORD_STRONG:= MesBlock2_Temp[(ParamNbRackString+1)*(KK-1)+JJ+1][ 95], Word_WEAK:= MesBlock2_Temp[(ParamNbRackString+1)*(KK-1)+JJ+1][96], 	SIGNED:=FALSE, FIX:=0 , SIZE:=2, VAR_OUT := MesDataExd.AX_RACK[CalrackNb].AX_RACKSTRING[JJ].MesMaxBalancingTime);

			END_IF
		END_IF


	END_FOR 

END_FOR


SUPER^.M_Read();
END_METHOD

METHOD M_StartStop
//////////////////
//  Start or stop BBMS via CAN bus   
/////////////////

VAR 
	// Method local variables (reinitialized at each cycle) 
		KK			: INT;

		CP_Start	: BOOL;
		CI_RPM		: BOOL;
		CI_BIR		: BOOL;
		CI_IDC1		: BOOL;
		CI_IDC2		: BOOL ; 
		CI_BS		: BOOL;
		CI_BST		: BOOL;
		CI_RSR		: BOOL;
		CI_FCR		: BOOL;
		CI_ESTP		: BOOL;
END_VAR

SUPER^.M_StartStop();
END_METHOD

METHOD M_StateManager
//////////////////
// Detect which is the state of the PCS system . 
/////////////////

VAR 
	// Method local variables (reinitialized at each cycle) 

	
END_VAR
MesDataExd.MesData.MesState 		:= 0 ; 

IF MesDataExd.MesSystemMode.8 THEN
	MesDataExd.MesData.MesState .2 := 1;
ELSIF MesDataExd.MesSystemMode.7 THEN
	MesDataExd.MesData.MesState .1 := 1;
ELSIF MesDataExd.MesSystemMode.6 THEN
	MesDataExd.MesData.MesState .0 := 1;
END_IF
	
SUPER^.M_StateManager() ;
END_METHOD

METHOD M_Write
VAR_INPUT
END_VAR
VAR
	InputAddr: WORD;
	RTCWord: ARRAY[1..6] OF BYTE;
	TriggerRTC: BOOL;
END_VAR
Trig_CmdCloseDC(CLK := IN_CmdCloseDC);
Trig_CmdOpenDC(CLK := IN_CmdOpenDC);
Trig_CmdReset(CLK := IN_CmdReset);

IF Trig_CmdCloseDC.Q THEN
	IN_CmdCloseDC := FALSE;
	AX_Cmd[1] := 16#0005;
END_IF
IF Trig_CmdOpenDC.Q THEN
	IN_CmdOpenDC := FALSE;
	AX_Cmd[1] := 16#0003;
END_IF
IF Trig_CmdReset.Q THEN			// lacth the fault date of events. WE HAVE TO CHECK FIRST THE FAULT BEFORE DOING IT/ 
	IN_CmdReset := FALSE;
	AX_Cmd[2] := 16#0050;
END_IF

Trig_Watchdog(CLK := CalLocalTimeStruct.wSecond MOD 5 = 0 );	// watchdog every 5 seconds . 
IF Trig_Watchdog.Q THEN
	AX_Cmd[3] := CalLocalTimeStruct.wSecond;
END_IF

AX_ModbusWrite[1]
(
	InputWord	:= AX_Cmd[1],
	sIPAddr 	:= ParamIpAddress,
	tTimeout 	:= ParamTimeout,
	nTCPport 	:= ParamTcpPort,
	nMBAddr 	:= 0,
	nUnitID 	:= ParamUnitID,
	WriteCmd 	:= Trig_CmdCloseDC.Q OR Trig_CmdOpenDC.Q AND MesDataExd.Mesdata.MesCP_Write ,
);




AX_ModbusWrite[2]
(
	InputWord	:= AX_Cmd[2],
	sIPAddr 	:= ParamIpAddress,
	tTimeout 	:= ParamTimeout,
	nTCPport 	:= ParamTcpPort,
	nMBAddr 	:= 1,
	nUnitID 	:= ParamUnitID,
	WriteCmd 	:= Trig_CmdReset.Q AND MesDataExd.Mesdata.MesCP_Write,
);

AX_ModbusWrite[3]	// Wa&tchdog 
(
	InputWord	:= AX_Cmd[3],
	sIPAddr 	:= ParamIpAddress,
	tTimeout 	:= ParamTimeout,
	nTCPport 	:= ParamTcpPort,
	nMBAddr 	:= 2,
	nUnitID 	:= ParamUnitID,
	WriteCmd 	:= Trig_Watchdog.Q AND MesDataExd.Mesdata.MesCP_Write,
);


// Write Datetime to BMS to keep same date . 
RTCWord[1] := WORD_TO_BYTE(2000 - CalLocalTimeStruct.wYear) ; 
RTCWord[2] :=  WORD_TO_BYTE(CalLocalTimeStruct.wMonth); 
RTCWord[3] := WORD_TO_BYTE(CalLocalTimeStruct.wDay); 
RTCWord[4] := WORD_TO_BYTE(CalLocalTimeStruct.wHour); 
RTCWord[5] := WORD_TO_BYTE(CalLocalTimeStruct.wMinute); 
RTCWord[6] := WORD_TO_BYTE(CalLocalTimeStruct.wSecond); 

TriggerRTC := CalLocalTimeStruct.wHour = 5 AND CalLocalTimeStruct.wMinute = 0 AND CalLocalTimeStruct.wSecond = 0 ; // Write dat once a day

A1_ModbusWriteRTC	// 
(   
	cbLength :=  SIZEOF(RTCWord ) ,
	pSrcAddr	:= ADR(RTCWord) , 
	nQuantity	:= 3 ,
	sIPAddr 	:= ParamIpAddress,
	tTimeout 	:= ParamTimeout,
	nTCPport 	:= ParamTcpPort,
	nMBAddr 	:= 0,
	nUnitID 	:= ParamUnitID,
	WriteCmd 	:=  (TriggerRTC) AND MesDataExd.Mesdata.MesCP_Write,
	Reset				:= CmdClearFault_G, 
);


	
SUPER^.M_Write();
END_METHOD

END_FUNCTION_BLOCK

// ---- 01_Equipement_Library/Batteries/FB_BAT_KP_MK1.TcPOU
FUNCTION_BLOCK FB_BAT_KP_MK1 EXTENDS FB_BAT_Base
// Code for the KorePower Mark1 battery system
// Architecture : 	MsBMS (1 - 40 racks per MsBMS)
//						Racks (2 - 17 modules per racks)
// 							Cells (32 per modules : 2P16S)

VAR_INPUT PERSISTENT
		ParamIpAddress 			: STRING 	:='192.168.127.133' ; 		(* IP¨Address*)
		ParamUnitID				: BYTE  	:= 1 ; 					(* Modbus Unit ID*)
		ParamTcpPort			: UINT 		:= 502;					(* Modbus TCP Port*)
	

END_VAR

VAR_INPUT
	//Child objects
	
	
		IN_CmdOpenDC						: BOOL;
		IN_CmdCloseDC 						: BOOL;
		
		MesDataExd							: BAT_KP;
END_VAR

VAR
	//M_ALARMMANAGEMENT VARIABLES//
	
		CalModbusWriteAlarm			: BOOL;		// Modbus Write alarm
		ComWarning					: BOOL;		// Aggregated Communication warning
		ComAlarm					: BOOL;		// Aggregated communication Alarm
	
		TON_BatteriesCharging		: TON ;
		TON_BatteriesDischarging	: TON ;
		
		
	//M_READ VARIABLES//
		ModbusRead802			: FB_ModbusRead;
		ModbusRead803_Fix		: FB_ModbusRead;
		
		MesModbusReadAlarm 		  	: ARRAY[1..2] OF BOOL ; 			// (NA) Modbus Read Alarm for all modbus frames		
		MesModbusReadAlarmRacks		: ARRAY[1..CstNbRack_BAT_G] OF ARRAY[1..2] OF BOOL ; 			// (NA) Modbus Read Alarm for all modbus frames
		
		
		// Au max, 40 strings, avec 32 registres : Je vais pouvoir faire 3 strings par requête (=96 reg/requetes) donc au max il y aura 13 requêtes
		ModbusRead803_Rep		: ARRAY[1..40] OF FB_ModbusRead;
		NbRead					: UDINT;
		
		StartAddr 				: UINT := 102;
	
		// Les blocks fixes du 804 ne sont jamais à la suite les uns des autres, donc il en faut au max 40.
		ModbusRead804_Fix		: ARRAY[1..40] OF FB_ModbusRead;
		// les blocs qui se répètent du 804 dépendent du nombre de modules par string : le nombre max est 17, avec 16 registres = 272 registres
		// je vais donc lire 112 registres 2 fois et 48 registres 1 fois
	
		                    	
		                    	
		MesBlock_802			: ARRAY[1..120] OF WORD;
		MesBlock_803_Fix		: ARRAY[1..120] OF WORD;
		MesBlock_803_Rep		: ARRAY[1..40] OF ARRAY[1..32*3] OF WORD;
		MesBlock_804_Fix		: ARRAY[1..40] OF ARRAY[1..48] OF WORD;
		                    	
		Cal_StartRead803_Fix	: UINT;
		Cal_StartRead804_Fix	: UINT;
	
	        
		MesChargeStatus			: UINT ; // temp charge status used before putting it in words
		MesIDState				: UINT ; // temp status used before putting it in words
		MesAHRtg_SF_802 		: REAL ; // Scale factor for charge capacity.
		MesWHRtg_SF_802 		: REAL ; // Scale factor for energy capacity.
		MesWChaDisChaMax_SF_802 : REAL ; // Scale factor for maximum charge and discharge rate.
		MesDisChaRte_SF_802 	: REAL ; // Scale factor for self discharge rate.
		MesSoC_SF_802 			: REAL ; // Scale factor for state of charge values.
		MesDoD_SF_802 			: REAL ; // Scale factor for depth of discharge.
		MesSoH_SF_802 			: REAL ; // Scale factor for state of health.
		MesV_SF_802 			: REAL ; // Scale factor for DC bus voltage.
		MesCellV_SF_802 		: REAL ; // Scale factor for cell voltage.
		MesA_SF_802 			: REAL ; // Scale factor for DC current.
		MesAMax_SF_802 			: REAL ; // Scale factor for instantaneous DC charge/discharge current.
		MesW_SF_802 			: REAL ; // Scale factor for AC power request.
		
		MesCellV_SF_803 		: REAL ; // Scale factor for cell voltage.
		MesModTmp_SF_803		: REAL ; // Scale factor for module temperatures.
		MesA_SF_803 			: REAL ; // Scale factor for string currents.
		MesSoH_SF_803 			: REAL ; // Scale factor for string state of health.
		MesSoC_SF_803 			: REAL ; // Scale factor for string state of charge.
		MesV_SF_803 			: REAL ; // Scale factor for string voltage.
	
		MesCellV_SF_804 		: REAL ; // Scale factor for cell voltage.
		MesModTmp_SF_804		: REAL ; // Scale factor for module temperatures.
		MesA_SF_804 			: REAL ; // Scale factor for string currents.
		MesSoH_SF_804 			: REAL ; // Scale factor for string state of health.
		MesSoC_SF_804 			: REAL ; // Scale factor for string state of charge.
		MesDoD_SF_804 			: REAL ; // Scale factor for string state of charge.
		MesV_SF_804 			: REAL ; // Scale factor for string voltage.

		                    	
	//M_WRITE VARIABLES //  	
		AX_Cmd	AT%Q* 			: ARRAY[1..3] OF WORD;
		AX_ModbusWrite			: ARRAY[1..4] OF FB_ModbusWriteSingleRegister;
		AX_bAlarmWrite			: ARRAY[1..4] OF BOOL;
		AX_uAlarmWrite			: ARRAY[1..4] OF UDINT ; 
		Trig_CmdOpenDC			: R_TRIG;
		Trig_CmdCloseDC			: R_TRIG;
		Trig_CmdReset			: R_TRIG;
	
	//M_STATEMANAGER VARIABLES//
	
	//M_INIT VARIABLES //
	//M_EVALUATE VARIABLES //
	
		
	
	//M_EXECUTE VARIABLES//
		
	//Test//	
		Xtest				: BOOL;
		xTestReal			: REAL;
		xTestReal1			: REAL;
		xTestInt			: INT;
		xTestWord			: WORD;
		
		
END_VAR

METHOD M_AlarmManagement
//////////////////
//  Battery Area  Alarm Management 
/////////////////

VAR 
	// Method local variables (reinitialized at each cycle) 
	FB_AlarmCodeManager 		: FB_AlarmCodeManager ; 
                            	
	KK							: UINT;				// For Loop 
	                 
END_VAR
//COMMUNICATION//
	CalModbusWriteAlarm := AX_bAlarmWrite[1] OR AX_bAlarmWrite[2] OR AX_bAlarmWrite[3] ; 
	
	ComWarning 			:= CalModbusWriteAlarm ;			// At least one modbus trame did not work
	ComAlarm			:= TRUE;						// All modbus trame did not work
	
	FOR KK:=1 TO 2 DO // nb of trame = 4
		ComWarning 	:= ComWarning OR MesModbusReadAlarm[KK] ;
		ComAlarm	:= ComAlarm AND MesModbusReadAlarm[KK];
	END_FOR
	
	FOR KK:=1 TO ParamNbRacks DO // nb of trame = 4
		ComWarning 	:= ComWarning OR MesModbusReadAlarmRacks[KK][1] OR MesModbusReadAlarmRacks[KK][2] ;
		ComAlarm	:= ComAlarm AND MesModbusReadAlarmRacks[KK][1] AND MesModbusReadAlarmRacks[KK][2];
	END_FOR	
	
	//Warning
	MesDataExd.MesData.MesWarningCom := ComWarning ; 
	//Alarm
	TON_ComAlarm(IN:= ComAlarm , PT:= ParamTempoComAlarm, Q=>MesDataExd.MesData.MesAlarmCom) ;	// Alarms if ALL TRAM MODBUS did not work and timeout of 15s
	


TON_ComAlarm(IN:= ComAlarm , PT:= ParamTempoComAlarm, Q=>MesDataExd.MesData.MesAlarmCom) ;	// Alarms if ALL TRAM MODBUS did not work and timeout of 15s
	



	FB_AlarmCodeManager(	
		bAlarm1			:= MesDataExd.MesData.MesAlarmCom, 									// Com alarm
		bAlarm2			:= FALSE,									// 
		bAlarm3			:= FALSE, 													//                  
		bAlarm4			:= FALSE, 													//                      
		bAlarm5			:= FALSE, 													//                 
		bAlarm6			:= FALSE, 													//          
		bAlarm7			:= FALSE, 													//          
		bAlarm8			:= FALSE, 													//          
		bAlarm9			:= FALSE,   												//         
		bAlarm10		:= FALSE,   												//         
		bAlarm11		:= FALSE,   												//          
		bAlarm12		:= FALSE, 													//  						                
		bAlarm13		:= FALSE, 													//  						                 
		bAlarm14		:= FALSE, 													//  						                 
		bAlarm15		:= FALSE, 													//  						
		wAlarmCode		=> MesDataExd.MesData.MesAlarmCode);


// WARNING CODE //
	FB_AlarmCodeManager(	
		bAlarm1			:= MesComWarning, 											// Communication warning 
		bAlarm2			:= FALSE, 													//
		bAlarm3			:= FALSE, 													//
		bAlarm4			:= FALSE, 													//      
		bAlarm5			:= FALSE, 													//      
		bAlarm6			:= FALSE, 													//      
		bAlarm7			:= FALSE, 													//      
		bAlarm8			:= FALSE,   												//         
		bAlarm9			:= FALSE,   												//         
		bAlarm10		:= FALSE,   												//         
		bAlarm11		:= FALSE,   												//         
		bAlarm12		:= FALSE,   												//         
		bAlarm13		:= FALSE,  													//         
		bAlarm14		:= FALSE,  													//         
		bAlarm15		:= FALSE,	    											// 
		wAlarmCode		=> MesDataExd.MesData.MesWarningCode);          
		


